# B&R Automation Studio project NAEUL004C00R13L518F00 (part 35)

#### Act_Main.st - Do Not Change!!!
```iecst
(** 2022-12-20 **)
ACTION Act_Background:

	a_tyAlmData[1]	:= tyAlmData;

	IF (bRstErr = TRUE) THEN

		tylocalAlm.Out.bErr		:= FALSE;
		tylocalAlm.Out.bWarning	:= FALSE;

		//Reset Warning
		memset(ADR(a_tyWarningCurrList) , 0 , SIZEOF(a_tyWarningCurrList));
		udiWarningMax	:=1;

		memset(ADR(tylocalAlm.Out.a_tyCurrList) , 0 , SIZEOF(tylocalAlm.Out.a_tyCurrList));
	//	memset(ADR(tylocalAlm.Out.a_sRecoveryList) , 0 , SIZEOF(tylocalAlm.Out.a_sRecoveryList));
		memset(ADR(tylocalAlm.Out.a_udiRecoveryList),0,SIZEOF(tylocalAlm.Out.a_udiRecoveryList));

		udiAlmCntr	:= 0;

		bAlmUpdt	:= FALSE;

	END_IF

	IF (bRstWarning = TRUE) THEN

		IF tylocalAlm.Out.bErr =FALSE AND tylocalAlm.Out.bWarning= TRUE THEN
			//Reset Warning
			memset(ADR(a_tyWarningCurrList) , 0 , SIZEOF(a_tyWarningCurrList));
			udiWarningMax	:=1;

			memset(ADR(tylocalAlm.Out.a_tyCurrList) , 0 , SIZEOF(tylocalAlm.Out.a_tyCurrList));
		//	memset(ADR(tylocalAlm.Out.a_sRecoveryList) , 0 , SIZEOF(tylocalAlm.Out.a_sRecoveryList));
			memset(ADR(tylocalAlm.Out.a_udiRecoveryList),0,SIZEOF(tylocalAlm.Out.a_udiRecoveryList));
			udiAlmCntr	:= 0;
			tylocalAlm.Out.bWarning := FALSE;
		END_IF

		bAlmUpdt	:= FALSE;

	END_IF

	IF bAlarmLog = TRUE  AND tylocalAlm.In.bStartupUISettingsLoadDone THEN

		IF (bAlmUpdt = FALSE) OR (tylocalAlm.Out.eStatus = Error) THEN

			tylocalAlm.Out.bInfo		:= FALSE;
			tylocalAlm.Out.bInfoLF		:= FALSE;
			iInfoCntr	:= 0;

			FOR udi := 1 TO c_udiAlarmCurrMax DO

				IF (a_tyAlmData[udi].udiRunTime <> a_udiRunTimeOld[udi]) AND a_tyAlmData[udi].udiCode <> 0
					AND ((a_tyAlmData[udi].eSeverity = AlmSeverityError ) ) THEN

					a_udiRunTimeOld[udi]	:= a_tyAlmData[udi].udiRunTime;

					bAlmUpdt	:= TRUE;

					udiAlmCntr	:= udiAlmCntr + 1;
					IF udiAlmCntr > c_udiAlarmCurrMax THEN
						udiAlmCntr	:= c_udiAlarmCurrMax;
					END_IF

					udiLogCntr	:= udiLogCntr + 1;
					IF udiLogCntr > c_udiAlarmCurrMax THEN
						udiLogCntr	:= c_udiAlarmCurrMax;
					END_IF

					fLogDTConvert(ADR(sDT) , tylocalAlm.In.dtCurrDT);

					IF a_tyAlmData[udi].udiCode < 10000 THEN
						udiErrorCode := a_tyAlmData[udi].udiCode;
					ELSE
						udiErrorCode := (a_tyAlmData[udi].udiCode - 10000) + (a_tyAlmData[udi].udiModuleNum);//*For HMI Text Group*
					END_IF

					//In this case, Program Name/Data Time/
					//Current List
					tylocalAlm.Out.a_tyCurrList[udiAlmCntr].eSeverity		:= a_tyAlmData[udi].eSeverity;
					tylocalAlm.Out.a_tyCurrList[udiAlmCntr].sDT				:= sDT;

					//To HMI Text Group
					tylocalAlm.Out.a_tyCurrList[udiAlmCntr].udiErrorCode	:= udiErrorCode;
					tylocalAlm.Out.a_tyCurrList[udiAlmCntr].bAlm			:= a_tyAlmData[udi].bAlm;

					//Recovery List
					tylocalAlm.Out.a_udiRecoveryList[udiAlmCntr]			:= udiErrorCode; //*For HMI Text Group **It will be the same procedure with the above**

					//History List
					memmove(ADR(a_tyHistoryList[2]) , ADR(a_tyHistoryList[1]) , SIZEOF(a_tyHistoryList[1]) * (c_udiAlarmHistoryMax - 1));

					a_tyHistoryList[1].sDT				:= sDT;
					a_tyHistoryList[1].udiModErrCode	:= a_tyAlmData[udi].udiCode;
					a_tyHistoryList[1].udiErrorCode		:= udiErrorCode;

					//Log List
					//					fLogAlmDispMsg(ADR(sAlmMsg) , tylocalAlm.In.dtCurrDT , a_tyAlmData[udi].sProgNm , a_tyAlmData[udi].udiCode , a_tyAlmData[udi].sAlmMsg); // *For Log files*
					//					a_sLogList[udiLogCntr]	:= sAlmMsg;
					a_sLogList[udiLogCntr]	:= CONCAT(a_sLogList[udiLogCntr] , '$r$n');

					//Severity
					IF a_tyAlmData[udi].eSeverity = AlmSeverityError THEN
						tylocalAlm.Out.bErr		:= TRUE;
					END_IF

					// Alarm warning
				ELSIF (( a_tyAlmData[udi].eSeverity = AlmSeverityWarning) AND  (a_tyAlmData[udi].udiCode <> 0 )) THEN

					//Used to compare
					memset(ADR(sWarningCompareMsg) , 0 , SIZEOF(sWarningCompareMsg));

					//					sWarningCompareMsg	:= CONCAT(sWarningCompareMsg , a_tyAlmData[udi].sProgNm);
					//					sWarningCompareMsg	:= CONCAT(sWarningCompareMsg , ' | ');
					//					sWarningID := UDINT_TO_STRING(a_tyAlmData[udi].udiCode);
					//					sWarningCompareMsg	:= CONCAT(sWarningCompareMsg , sWarningID);
					//					sWarningCompareMsg	:= CONCAT(sWarningCompareMsg , ' | ');
					////					sWarningCompareMsg	:= CONCAT(sWarningCompareMsg , a_tyAlmData[udi].sAlmMsg);
					//
					//					//Checking whether it is recorded in the alarm list
					//					FOR udi1 := 0 TO  udiWarningMax DO
					//						WarningListOccur := (memcmp(ADR(sWarningCompareMsg),ADR(a_tyWarningCurrList[udi1].sMsg),SIZEOF(sWarningCompareMsg) )= 0);
					//
					//						IF WarningListOccur THEN
					//							EXIT;
					//						END_IF
					//
					//					END_FOR

					//IF warning message is no recorded in alarm list
					IF 	WarningListOccur =FALSE THEN

						bAlmUpdt	:= TRUE;
						udiWarningMax := udiWarningMax +1;

						udiAlmCntr	:= udiAlmCntr + 1;

						IF udiAlmCntr > c_udiAlarmCurrMax THEN
							udiAlmCntr	:= c_udiAlarmCurrMax;
						END_IF

						udiRecorded[udiWarningMax-1]:= udi;

						udiLogCntr	:= udiLogCntr + 1;

						IF udiLogCntr > c_udiAlarmCurrMax THEN
							udiLogCntr	:= c_udiAlarmCurrMax;
						END_IF

						//Warning List
						//						a_tyWarningCurrList[udiWarningMax-1].sMsg		:= sWarningCompareMsg;

						fLogDTConvert(ADR(sDT) , tylocalAlm.In.dtCurrDT);
						udiErrorCode := (a_tyAlmData[udi].udiCode - 10000) + a_tyAlmData[udi].udiModuleNum; //*For HMI Text Group*

						//Current List
						tylocalAlm.Out.a_tyCurrList[udiAlmCntr].eSeverity		:= a_tyAlmData[udi].eSeverity;
						tylocalAlm.Out.a_tyCurrList[udiAlmCntr].sDT				:= sDT;
						tylocalAlm.Out.a_tyCurrList[udiAlmCntr].udiModErrCode	:= a_tyAlmData[udi].udiCode;

						//To HMI Text Group
						tylocalAlm.Out.a_tyCurrList[udiAlmCntr].udiErrorCode	:= udiErrorCode;
						tylocalAlm.Out.a_tyCurrList[udiAlmCntr].bWarning		:= a_tyAlmData[udi].bWarning;

						//Recovery List
						//						tylocalAlm.Out.a_sRecoveryList[udiAlmCntr]	 	:= a_tyAlmData[udi].sRcyMsg;
						tylocalAlm.Out.a_udiRecoveryList[udiAlmCntr]	:= udiErrorCode;

						//History List
						memmove(ADR(a_tyHistoryList[2]) , ADR(a_tyHistoryList[1]) , SIZEOF(a_tyHistoryList[1]) * (c_udiAlarmHistoryMax - 1));

						a_tyHistoryList[1].sDT				:= sDT;
						a_tyHistoryList[1].udiModErrCode	:= a_tyAlmData[udi].udiCode;
						a_tyHistoryList[1].udiErrorCode		:= udiErrorCode;

						//Log List
						//Info Message
						//						fLogAlmDispMsg(ADR(sWarningMsg) , tylocalAlm.In.dtCurrDT , a_tyAlmData[udi].sProgNm , a_tyAlmData[udi].udiCode , a_tyAlmData[udi].sAlmMsg);

						a_sLogList[udiLogCntr]	:= sWarningMsg;
						a_sLogList[udiLogCntr]	:= CONCAT(a_sLogList[udiLogCntr] , '$r$n');

						tylocalAlm.Out.bWarning	:= TRUE;

					END_IF

					// Show Info Message
				ELSIF  ((a_tyAlmData[udi].udiCode <> 0) AND (a_tyAlmData[udi].eSeverity = AlmSeverityInfo)) THEN

					iInfoCntr	:= iInfoCntr + 1;

					IF iInfoCntr = 1 THEN

						IF a_tyAlmData[udi].udiModuleNum = 3901 AND a_tyAlmData[udi].bAlm THEN //Identify Leader Follower Inforamtion

							tylocalAlm.Out.bInfoLF	:= TRUE;
							tylocalAlm.Out.bInfo	:= TRUE;

						ELSE
							tylocalAlm.Out.bInfoLF	:= FALSE;
							tylocalAlm.Out.bInfo	:= TRUE;
						END_IF

					ELSIF iInfoCntr = 2 THEN
						//						tylocalAlm.sInfoMsg	:= CONCAT(tylocalAlm.sInfoMsg , '$r$n$r$n');
						//						tylocalAlm.sInfoMsg	:= CONCAT(tylocalAlm.sInfoMsg , a_tyAlmData[udi].sAlmMsg);

					END_IF

				END_IF

			END_FOR

		ELSE

			tylocalAlm.In.eAct	:= AlarmActAppendLogWriteHistory;
			IF tylocalAlm.Out.eStatus = Done AND tylocalAlm.Out.eStat = AlarmActAppendLogWriteHistory THEN
				tylocalAlm.In.eAct		:= AlarmActIdle;
				bAlmUpdt	:= FALSE;
				udiLogCntr	:= 0;
			END_IF

		END_IF

	END_IF
	//**** Background Running Done*****

	//Delete Old Alarm Log File for 24 hours After Machine is Continuous Running 30 Days.
	fbDlyTmr(IN := TRUE);
	IF fbDlyTmr.Q THEN
		fbDeleteLogTmr (IN := TRUE);
		IF fbDeleteLogTmr.Q AND eStatus <> Busy THEN
			p_eAct := AlarmActDeleteOldLog;
			IF eStat = AlarmActDeleteOldLog AND eStatus = Done THEN
				p_eAct := AlarmActIdle;
				fbDlyTmr (IN := FALSE);
				fbDeleteLogTmr (IN := FALSE);
			END_IF
		END_IF
	END_IF

	//Reset Done
	IF tylocalAlm.Out.eStatus = Done AND tylocalAlm.In.eAct = AlarmActIdle THEN
		tylocalAlm.Out.eStat	:= AlarmActIdle;
	END_IF

	//Set tylocalAlm.In.eAct
	IF tylocalAlm.Out.eStatus = Idle THEN
		tylocalAlm.Out.eStat	:= tylocalAlm.In.eAct;
	END_IF
	//Main
	CASE tylocalAlm.Out.eStat OF

		AlarmActIdle:
			IF tylocalAlm.Out.eStatus <> Idle THEN	//Reset Data
				//Private
				fbDirCreate1(bEn := FALSE);
				fbDirCreate2(bEn := FALSE);
				fbFileOldDel1(bEn := FALSE);
				fbFileRead1(bEn := FALSE);
				fbFileAppend1(bEn := FALSE);
				fbFileWrite1(bEn := FALSE);
				usiStep	:= 0;

				tylocalAlm.Out.bHistoryFileNotFound	:= FALSE;
				udiWriteLogCntr			:= 1;

				sStatTxt	:= a_sStatText[tylocalAlm.Out.eStat];

			END_IF

			tylocalAlm.Out.eStatus	:= Idle;

		AlarmActCreateDir:
			IF tylocalAlm.Out.eStatus = Idle OR tylocalAlm.Out.eStatus = Busy THEN

				tylocalAlm.Out.eStatus	:= Busy;

				sStatTxt	:= a_sStatText[tylocalAlm.Out.eStat];

				CASE usiStep OF
					0:
						fbDirCreate1(bEn := TRUE);
						IF fbDirCreate1.udiStatus = 0 THEN
							usiStep	:= 1;
						ELSIF fbDirCreate1.udiStatus < 65534 THEN
							tylocalAlm.Out.eStatus		:= Error;

							IF fbDirCreate1.udiStatus = 1908 THEN
								udiStatus	:= 5051;	//Create User Directory Error
							ELSE
								udiStatus	:= fbDirCreate1.udiStatus;
							END_IF
						END_IF

					1:
						fbDirCreate2(bEn := TRUE);
						IF fbDirCreate2.udiStatus = 0 THEN
							tylocalAlm.Out.eStatus	:= Done;
						ELSIF fbDirCreate2.udiStatus < 65534 THEN
							tylocalAlm.Out.eStatus		:= Error;

							IF fbDirCreate2.udiStatus = 1908 THEN
								udiStatus	:= 5052;	//Create Alarm Directory Error
							ELSE
								udiStatus	:= fbDirCreate2.udiStatus;
							END_IF
						END_IF

				END_CASE

			END_IF

		AlarmActDeleteOldLog:
			IF tylocalAlm.Out.eStatus = Idle OR tylocalAlm.Out.eStatus = Busy THEN

				tylocalAlm.Out.eStatus	:= Busy;

				sStatTxt	:= a_sStatText[tylocalAlm.Out.eStat];

				fbFileOldDel1.dtDTNow			:= tylocalAlm.In.dtCurrDT;
				fbFileOldDel1.udiFileKeepDay	:= tylocalAlm.In.udiFileKeepDay;
				fbFileOldDel1(bEn := TRUE);
				IF fbFileOldDel1.udiStatus = 0 THEN
					tylocalAlm.Out.eStatus	:= Done;
				ELSIF fbFileOldDel1.udiStatus < 65534 THEN
					tylocalAlm.Out.eStatus		:= Error;

					IF fbFileOldDel1.udiStatus = 1910 THEN
						udiStatus	:= 5053;	//Get Directory Info Error While Deleting Old Log
					ELSIF fbFileOldDel1.udiStatus = 1911 THEN
						udiStatus	:= 5054;	//Directory Read Error While Deleting Old Log
					ELSIF fbFileOldDel1.udiStatus = 1912 THEN
						udiStatus	:= 5055;	//File Delete Error While Deleting Old Log
					ELSE
						udiStatus	:= fbFileOldDel1.udiStatus;
					END_IF
				END_IF

			END_IF

		AlarmActReadHistory:
			IF tylocalAlm.Out.eStatus = Idle OR tylocalAlm.Out.eStatus = Busy THEN

				tylocalAlm.Out.eStatus	:= Busy;

				sStatTxt	:= a_sStatText[tylocalAlm.Out.eStat];

				fbFileRead1(bEn := TRUE);
				IF fbFileRead1.udiStatus = 0 THEN
					tylocalAlm.Out.eStatus	:= Done;
				ELSIF fbFileRead1.udiStatus < 65534 THEN
					tylocalAlm.Out.eStatus		:= Error;

					IF fbFileRead1.udiStatus = 1900 THEN
						udiStatus	:= 5056;	//File Open Error While Reading Alarm History
					ELSIF fbFileRead1.udiStatus = 1902 THEN
						udiStatus	:= 5057;	//File Read Error While Reading Alarm History
					ELSIF fbFileRead1.udiStatus = 1904 THEN
						udiStatus	:= 5058;	//File Close Error While Reading Alarm History
					ELSIF fbFileRead1.udiStatus = 1915 THEN
						tylocalAlm.Out.eStatus					:= Done;
						tylocalAlm.Out.bHistoryFileNotFound	:= TRUE;
					ELSE
						udiStatus	:= fbFileRead1.udiStatus;
					END_IF
				END_IF

			END_IF

		AlarmActWriteHistory:
			IF tylocalAlm.Out.eStatus = Idle OR tylocalAlm.Out.eStatus = Busy THEN

				tylocalAlm.Out.eStatus	:= Busy;

				sStatTxt	:= a_sStatText[tylocalAlm.Out.eStat];

				fbFileWrite1(bEn := TRUE);
				IF fbFileWrite1.udiStatus = 0 THEN
					tylocalAlm.Out.eStatus	:= Done;
				ELSIF fbFileWrite1.udiStatus < 65534 THEN
					tylocalAlm.Out.eStatus		:= Error;

					IF fbFileWrite1.udiStatus = 1900 THEN
						udiStatus	:= 5059;	//File Open Error While Writing Alarm History
					ELSIF fbFileWrite1.udiStatus = 1901 THEN
						udiStatus	:= 5060;	//File Create Error While Writing Alarm History
					ELSIF fbFileWrite1.udiStatus = 1903 THEN
						udiStatus	:= 5061;	//File Write Error While Writing Alarm History
					ELSIF fbFileWrite1.udiStatus = 1904 THEN
						udiStatus	:= 5062;	//File Close Error While Writing Alarm History
					ELSIF fbFileWrite1.udiStatus = 1914 THEN
						udiStatus	:= 5063;	//Directory Does Not Exist While Writing Alarm History
					ELSE
						udiStatus	:= fbFileWrite1.udiStatus;
					END_IF
				END_IF

			END_IF

		AlarmActAppendLog:
			IF tylocalAlm.Out.eStatus = Idle OR tylocalAlm.Out.eStatus = Busy THEN

				tylocalAlm.Out.eStatus	:= Busy;

				sStatTxt	:= a_sStatText[tylocalAlm.Out.eStat];

				dtCurrDTTemp			:= tylocalAlm.In.dtCurrDT;
				fbFileAppend1.sFile		:= DT_TO_STRING(dtCurrDTTemp);
				fbFileAppend1.sFile		:= MID(fbFileAppend1.sFile , 10 , 4);
				fbFileAppend1.sFile		:= CONCAT('ALARM_' , fbFileAppend1.sFile);
				fbFileAppend1.sFile		:= CONCAT(fbFileAppend1.sFile , '.dat');

				fbFileAppend1.p_Src		:= ADR(a_sLogList[udiWriteLogCntr]);
				fbFileAppend1.udiLen	:= LEN(a_sLogList[udiWriteLogCntr]);

				fbFileAppend1(bEn := TRUE);
				IF fbFileAppend1.udiStatus = 0 THEN
					IF udiWriteLogCntr >= udiLogCntr THEN
						tylocalAlm.Out.eStatus	:= Done;
					ELSE
						udiWriteLogCntr	:= udiWriteLogCntr + 1;
						fbFileAppend1(bEn := FALSE);
					END_IF

				ELSIF fbFileAppend1.udiStatus < 65534 THEN
					tylocalAlm.Out.eStatus		:= Error;

					IF fbFileAppend1.udiStatus = 1900 THEN
						udiStatus	:= 5064;	//File Open Error While Writing Alarm Log
					ELSIF fbFileAppend1.udiStatus = 1901 THEN
						udiStatus	:= 5065;	//File Create Error While Writing Alarm Log
					ELSIF fbFileAppend1.udiStatus = 1913 THEN
						udiStatus	:= 5066;	//Get File Info Error While Writing Alarm Log
					ELSIF fbFileAppend1.udiStatus = 1903 THEN
						udiStatus	:= 5067;	//File Write Error While Writing Alarm Log
					ELSIF fbFileAppend1.udiStatus = 1904 THEN
						udiStatus	:= 5068;	//File Close Error While Writing Alarm Log
					ELSIF fbFileAppend1.udiStatus = 1914 THEN
						udiStatus	:= 5069;	//Directory Does Not Exist While Writing Alarm Log
					ELSE
						udiStatus	:= fbFileAppend1.udiStatus;
					END_IF
				END_IF

			END_IF

		AlarmActAppendLogWriteHistory:
			IF tylocalAlm.Out.eStatus = Idle OR tylocalAlm.Out.eStatus = Busy THEN

				tylocalAlm.Out.eStatus	:= Busy;

				sStatTxt	:= a_sStatText[tylocalAlm.Out.eStat];

				dtCurrDTTemp			:= tylocalAlm.In.dtCurrDT;
				fbFileAppend1.sFile		:= DT_TO_STRING(dtCurrDTTemp);
				fbFileAppend1.sFile		:= MID(fbFileAppend1.sFile , 10 , 4);
				fbFileAppend1.sFile		:= CONCAT('ALARM_' , fbFileAppend1.sFile);
				fbFileAppend1.sFile		:= CONCAT(fbFileAppend1.sFile , '.dat');

				fbFileAppend1.p_Src		:= ADR(a_sLogList[udiWriteLogCntr]);
				fbFileAppend1.udiLen	:= LEN(a_sLogList[udiWriteLogCntr]);

				fbFileAppend1(bEn := TRUE);
				fbFileWrite1(bEn := TRUE);

				IF (fbFileAppend1.udiStatus = 0) AND (udiWriteLogCntr >= udiLogCntr) AND fbFileWrite1.udiStatus = 0 THEN
					tylocalAlm.Out.eStatus	:= Done;

				ELSIF fbFileAppend1.udiStatus = 0 AND udiWriteLogCntr < udiLogCntr THEN
					udiWriteLogCntr	:= udiWriteLogCntr + 1;
					fbFileAppend1(bEn := FALSE);

				ELSIF fbFileWrite1.udiStatus > 0 AND fbFileWrite1.udiStatus < 65534 THEN
					tylocalAlm.Out.eStatus		:= Error;

					IF fbFileWrite1.udiStatus = 1900 THEN
						udiStatus	:= 5070;	//File Open Error While Writing Alarm History
					ELSIF fbFileWrite1.udiStatus = 1901 THEN
						udiStatus	:= 5071;	//File Create Error While Writing Alarm History
					ELSIF fbFileWrite1.udiStatus = 1903 THEN
						udiStatus	:= 5072;	//File Write Error While Writing Alarm History
					ELSIF fbFileWrite1.udiStatus = 1904 THEN
						udiStatus	:= 5073;	//File Close Error While Writing Alarm History
					ELSIF fbFileWrite1.udiStatus = 1914 THEN
						udiStatus	:= 5074;	//Directory Does Not Exist While Writing Alarm History
					ELSE
						udiStatus	:= fbFileWrite1.udiStatus;
					END_IF

				ELSIF fbFileAppend1.udiStatus > 0 AND fbFileAppend1.udiStatus < 65534 THEN
					tylocalAlm.Out.eStatus		:= Error;

					IF fbFileAppend1.udiStatus = 1900 THEN
						udiStatus	:= 5075;	//File Open Error While Writing Alarm Log
					ELSIF fbFileAppend1.udiStatus = 1901 THEN
						udiStatus	:= 5076;	//File Create Error While Writing Alarm Log
					ELSIF fbFileAppend1.udiStatus = 1913 THEN
						udiStatus	:= 5077;	//Get File Info Error While Writing Alarm Log
					ELSIF fbFileAppend1.udiStatus = 1903 THEN
						udiStatus	:= 5078;	//File Write Error While Writing Alarm Log
					ELSIF fbFileAppend1.udiStatus = 1904 THEN
						udiStatus	:= 5079;	//File Close Error While Writing Alarm Log
					ELSIF fbFileAppend1.udiStatus = 1914 THEN
						udiStatus	:= 5080;	//Directory Does Not Exist While Writing Alarm Log
					ELSE
						udiStatus	:= fbFileAppend1.udiStatus;
					END_IF
				END_IF

			END_IF

		AlarmActResetHistory:
			IF tylocalAlm.Out.eStatus = Idle OR tylocalAlm.Out.eStatus = Busy THEN

				tylocalAlm.Out.eStatus	:= Busy;

				sStatTxt	:= a_sStatText[tylocalAlm.Out.eStat];

				memset(ADR(a_tyHistoryList) , 0 , SIZEOF(a_tyHistoryList));

				fbFileWrite1(bEn := TRUE);
				IF fbFileWrite1.udiStatus = 0 THEN
					tylocalAlm.Out.eStatus	:= Done;
				ELSIF fbFileWrite1.udiStatus < 65534 THEN
					tylocalAlm.Out.eStatus		:= Error;

					IF fbFileWrite1.udiStatus = 1900 THEN
						udiStatus	:= 5081;	//File Open Error While Resetting Alarm History
					ELSIF fbFileWrite1.udiStatus = 1901 THEN
						udiStatus	:= 5082;	//File Create Error While Resetting Alarm History
					ELSIF fbFileWrite1.udiStatus = 1903 THEN
						udiStatus	:= 5083;	//File Write Error While Resetting Alarm History
					ELSIF fbFileWrite1.udiStatus = 1904 THEN
						udiStatus	:= 5084;	//File Close Error While Resetting Alarm History
					ELSIF fbFileWrite1.udiStatus = 1914 THEN
						udiStatus	:= 5085;	//Directory Does Not Exist While Resetting Alarm History
					ELSE
						udiStatus	:= fbFileWrite1.udiStatus;
					END_IF
				END_IF

			END_IF

		AlarmActBGStartLog:
			IF tylocalAlm.Out.eStatus = Idle OR tylocalAlm.Out.eStatus = Busy THEN

				sStatTxt	:= a_sStatText[tylocalAlm.Out.eStat];

				bAlarmLog	:= TRUE;
				tylocalAlm.Out.eStatus		:= Done;

			END_IF

		AlarmActBGStopLog:
			IF tylocalAlm.Out.eStatus = Idle OR tylocalAlm.Out.eStatus = Busy THEN

				sStatTxt	:= a_sStatText[tylocalAlm.Out.eStat];

				bAlarmLog	:= FALSE;
				tylocalAlm.Out.eStatus		:= Done;

			END_IF

	END_CASE

	END_CASE
END_ACTION
```

#### Act_Alarm.st - Do Not Change!!!
```iecst
(** 2019-03-25 **)
ACTION Act_Alarm:
	IF tylocalAlm.In.udiRstErr <> udiRstErrOld THEN
		bRstErr			:= TRUE;
		udiRstErrOld	:= tylocalAlm.In.udiRstErr;
	ELSE
		bRstErr			:= FALSE;
	END_IF

	//Checking which Warning is clear
	IF a_tyWarningCurrList[1].sMsg <> '' AND p_tyLinkLibVerAlmData.udiCode = 0 THEN

		FOR udi2 := 1 TO (udiWarningMax-1) DO
			udiRecorded1:= udiRecorded[udi2];
			IF 	(pa_tyAlmData[udiRecorded1].eSeverity =  AlmSeverityNA) AND udiRecorded1<> 0 THEN
				bRstWarning := TRUE;
				EXIT;
			ELSE
				bRstWarning := FALSE;
			END_IF

		END_FOR
	ELSE
		bRstWarning := FALSE;
	END_IF

	//Reset Error
	IF (tylocalAlm.Out.eStatus = Error) AND bRstErr THEN
		tylocalAlm.In.eAct	:= AlarmActIdle;
		tylocalAlm.Out.eStat	:= AlarmActIdle;
	END_IF

	//Error
	IF EDGEPOS(tylocalAlm.Out.eStatus = Error) THEN

		tyAlmData.udiCode				:= udiStatus;
		tyAlmData.eSeverity				:= AlmSeverityError;
		tyAlmData.udiRunTime			:= tyAlmData.udiRunTime + 1;
		tyAlmData.bAlm					:= TRUE;
		tyAlmData.udiModuleNum  		:= udiModuleNum;
		g_tyAlmProgNm.sAlarmProgNm		:= g_tyNtParamCurr.sAlmProgNm;

		//Get Error Message
		IF tyAlmData.udiCode < 10000 OR tyAlmData.udiCode > 10099 THEN
			tyAlmData.sAlmMsg	:= 'Unknown';
			tyAlmData.sRcyMsg	:= 'Unknown';
		ELSE
			tyAlmData.sAlmMsg	:= a_tyAlmText[tyAlmData.udiCode].sAlmText;
			tyAlmData.sRcyMsg	:= a_tyAlmText[tyAlmData.udiCode].sRcyText;
		END_IF

		sStatTxt	:= tyAlmData.sAlmMsg;
	ELSIF bRstErr AND (tyAlmData.udiCode <> 0) THEN

		tyAlmData.udiCode	:= 0;
		tyAlmData.eSeverity	:= AlmSeverityNA;
		tyAlmData.bAlm			:= FALSE;
		sStatTxt	:= a_sStatText[tylocalAlm.Out.eStat];

	END_IF

END_ACTION
```

#### InputRef.var - Do Not Change!!!
```iecst
(*2019-03-25*)
(**)
(*General*)
VAR
	p_udiCurrMax : REFERENCE TO UDINT;
	p_udiHistoryMax : REFERENCE TO UDINT;
END_VAR
(**)
VAR
	p_eAct : REFERENCE TO eAlarmAction;
	p_udiRstErr : REFERENCE TO UDINT;
END_VAR
(**)
(*Configuration*)
VAR
	p_dtCurrDT : REFERENCE TO DATE_AND_TIME;
	pa_tyAlmData : REFERENCE TO ARRAY[1..c_udiAlarmCurrMax] OF tyAlmDat;
	p_udiFileKeepDay : REFERENCE TO UDINT;
	p_sProgNm : REFERENCE TO STRING[15];
	p_bNtSettingsLoadDone : REFERENCE TO BOOL;
	p_bStartupUISettingsLoadDone : REFERENCE TO BOOL;
END_VAR
```

#### Local.var - Do Not Change!!!
```iecst
(*2019-05-09*)
(**)
(*Local Action, State & Status*)
VAR
	udiStatus : UDINT := 0;
	sStatTxt : STRING[200] := '';
	a_sStatText : ARRAY[0..50] OF STRING[200] := ['Idling','Creating Directory','Deleting Old Alarm Log File','Reading History File','Writing History File','Appending Alarm Log File','Appending Alarm Log File & Writing History File','Resetting History','Background Start Alarm Log','Background Stop Alarm Log',41('')];
END_VAR
(**)
(*Local Alarm*)
VAR
	tyAlmData : tyAlmDat;
	tylocalAlm : tyAlarm;
	a_tyAlmData : ARRAY[1..c_udiAlarmCurrMax] OF tyAlmDat;
END_VAR
(**)
(*Local Output*)
VAR
	bErr : BOOL;
	bWarning : BOOL;
	a_tyCurrList : ARRAY[1..c_udiAlarmCurrMax] OF tyAlarmCurr;
	a_udiRecoveryList : ARRAY[1..c_udiAlarmCurrMax] OF UDINT;
	a_sHistoryList : ARRAY[1..c_udiAlarmHistoryMax] OF STRING[200];
	bInfo : BOOL;
	sInfoMsg : STRING[200];
	bHistoryFileNotFound : BOOL;
	bInfoLF : BOOL := FALSE;
END_VAR
(**)
(*Local Input*)
VAR
	udiRstErr : UDINT := 0;
	dtCurrDT : DATE_AND_TIME;
	udiFileKeepDay : UDINT := 30;
	sProgNm : STRING[15] := 'Alarm';
	bNtSettingsLoadDone : BOOL := TRUE;
END_VAR
(**)
(*Local*)
VAR
	bRstErr : BOOL;
	udiRstErrOld : UDINT;
	bInitDone : BOOL;
	bInitialDone : BOOL;
	bAlarmLog : BOOL;
	usiStep : USINT;
	udi : UDINT;
	iInfoCntr : INT;
	sAlmMsg : STRING[300];
	udiAlmCntr : UDINT;
	udiAlmRecvryCntr : UDINT;
	udiLogCntr : UDINT;
	udiWriteLogCntr : UDINT;
	a_sLogList : ARRAY[1..c_udiAlarmCurrMax] OF STRING[200];
	bAlmUpdt : BOOL;
	dtCurrDTTemp : DATE_AND_TIME;
	a_udiRunTimeOld : ARRAY[1..c_udiAlarmCurrMax] OF UDINT;
	fbDirCreate1 : fbDirCreate;
	fbDirCreate2 : fbDirCreate;
	fbFileAppend1 : fbFileFullAppend;
	fbFileOldDel1 : fbFileOldDel;
	fbFileRead1 : fbFileFullRead;
	fbFileWrite1 : fbFileFullWrite;
	udi1 : UDINT;
	udi2 : UDINT;
	udiRecorded : ARRAY[1..c_udiAlarmCurrMax] OF UDINT;
	udiRecorded1 : UDINT;
	bRstWarning : BOOL;
	udiWarningMax : UDINT := 1;
	sWarningMsg : STRING[300];
	sWarningID : STRING[80] := '';
	sWarningCompareMsg : STRING[300];
	a_tyWarningCurrList : ARRAY[1..c_udiAlarmCurrMax] OF tyAlarmCurr;
	a_tyHistoryList : ARRAY[1..c_udiAlarmHistoryMax] OF tyHistory;
	WarningListOccur : BOOL := TRUE;
	udiErrorCode : UDINT;
	sDT : STRING[80];
	sLogString : STRING[200];
	udiModuleNum : UDINT := 5051;
END_VAR
```

#### Act_InputConfig.st - not listed in the package file held
```iecst
ACTION Act_InputConfig:

	tylocalAlm.In.udiRstErr					 := g_tyRstErrOut.udiRstErr;
	tylocalAlm.In.eAct					 	 := g_tyStartUp.eAlarmAct;
	tylocalAlm.In.dtCurrDT  			  	 := g_tyTime.dtCurrDT;
	tylocalAlm.In.udiFileKeepDay		 	 := g_tyNtParamCurr.udiAlmFileKeepDay;
	tylocalAlm.In.sProgNm					 := g_tyNtParamCurr.sAlmProgNm;
	tylocalAlm.In.bStartupUISettingsLoadDone := g_tyStartUp.bUISettingsLoadDone;

	//Index 1 For Internal Use
	a_tyAlmData[2]		:= g_tyUsrFolder.tyAlmData;
	a_tyAlmData[3]		:= g_tyLibVer.tyAlmData;
	a_tyAlmData[4]		:= g_tyTime.tyAlmData;
	a_tyAlmData[5]		:= g_tyTime.tyAlmData1;
	a_tyAlmData[6]		:= g_tyHWInfo.tyAlmData;
	a_tyAlmData[7]		:= g_tyProdRcp.tyAlmData;
	a_tyAlmData[8]		:= g_tyMpProdRcp.tyAlmData;
	a_tyAlmData[9]		:= g_tyMagRcp.tyAlmData;
	a_tyAlmData[10]		:= g_tyMcParam.tyAlmData;
	a_tyAlmData[11]		:= g_tyNtParam.tyAlmData;
	a_tyAlmData[12]		:= g_tyUsrMgmt.tyAlmData;
	a_tyAlmData[13]		:= g_tyBuffer1.tyAlmData;
	a_tyAlmData[14]		:= g_tyBuffer2.tyAlmData;
	a_tyAlmData[15]		:= g_tyBuffer3.tyAlmData;
	a_tyAlmData[16]		:= g_tyUSSMEMAA.tyAlmData;
	a_tyAlmData[17]		:= g_tyUSSMEMAB.tyAlmData;
	a_tyAlmData[18]		:= g_tyUSSMEMA1.tyAlmData;
	a_tyAlmData[19]		:= g_tyUSSMEMA2.tyAlmData;
	a_tyAlmData[20]		:= g_tyUSSMEMA3.tyAlmData;
	a_tyAlmData[21]		:= g_tyDSSMEMA1.tyAlmData;
	a_tyAlmData[22]		:= g_tyDSSMEMA2.tyAlmData;
	a_tyAlmData[23]		:= g_tyDSSMEMA3.tyAlmData;
	a_tyAlmData[24]		:= g_tyInShutter.tyAlmData;
	a_tyAlmData[25]		:= g_tyOutShutter.tyAlmData;
	a_tyAlmData[26]		:= g_tyStopperA.tyAlmData;
	a_tyAlmData[27]		:= g_tyStopperB.tyAlmData;
	a_tyAlmData[28]		:= g_tyPshrConv.tyAlmData;
	a_tyAlmData[29]		:= g_tyMagConv1.tyAlmData;
	a_tyAlmData[30]		:= g_tyMagConv2.tyAlmData;
	a_tyAlmData[31]		:= g_tyMagConv3.tyAlmData;
	a_tyAlmData[32]	:= g_tyAWOpen.tyAlmData;
	a_tyAlmData[33]	:= g_tyAWOpen.tyAlmData1;
	a_tyAlmData[34]	:= g_tyAWOpen.tyAlmData2;
	a_tyAlmData[35]	:= g_tyAWOpen.tyAlmData3;
	a_tyAlmData[36]	:= g_tyTrav.tyAlmData;
	a_tyAlmData[37]	:= g_tyTrav.tyAlmData1;
	a_tyAlmData[38]	:= g_tyTrav.tyAlmData2;
	a_tyAlmData[39]	:= g_tyTrav.tyAlmData3;
	a_tyAlmData[40]	:= g_tyLifterBtm.tyAlmData;
	a_tyAlmData[41]	:= g_tyLifterBtm.tyAlmData1;
	a_tyAlmData[42]	:= g_tyLifterBtm.tyAlmData2;
	a_tyAlmData[43]	:= g_tyLifterBtm.tyAlmData3;
	a_tyAlmData[44]	:= g_tyDI.tyAlmData1;
	a_tyAlmData[45]	:= g_tyDI.tyAlmData2;
	a_tyAlmData[46]	:= g_tyDI.tyAlmData3;
	a_tyAlmData[47]	:= g_tyDI.tyAlmData4;
	a_tyAlmData[48]	:= g_tyAGVMag1.tyAlmData;
	a_tyAlmData[49]	:= g_tyAGVMag2.tyAlmData;
	a_tyAlmData[50]	:= g_tyAGVMag3.tyAlmData;
	a_tyAlmData[51]	:= g_tyHermes.tyAlmData;
	a_tyAlmData[52]	:= g_tyUSHermesA.tyAlmData;
	a_tyAlmData[53]	:= g_tyUSHermesA.tyAlmData1;
	a_tyAlmData[54]	:= g_tyUSHermesA.tyAlmData2;
	a_tyAlmData[55]	:= g_tyUSHermesA.tyAlmData3;
	a_tyAlmData[56]	:= g_tyUSHermesA.tyAlmData4;
	a_tyAlmData[57]	:= g_tyUSHermesAInfoData;
	a_tyAlmData[58]	:= g_tyUSHermesB.tyAlmData;
	a_tyAlmData[59]	:= g_tyUSHermesB.tyAlmData1;
	a_tyAlmData[60]	:= g_tyUSHermesB.tyAlmData2;
	a_tyAlmData[61]	:= g_tyUSHermesB.tyAlmData3;
	a_tyAlmData[62]	:= g_tyUSHermesB.tyAlmData4;
	a_tyAlmData[63]	:= g_tyUSHermesBInfoData;
	a_tyAlmData[64]	:= g_tyRmtHermes.tyAlmData;
	a_tyAlmData[65]	:= g_tyRmtHermes.tyAlmData1;
	a_tyAlmData[66]	:= g_tyRmtHermes.tyAlmData2;
	a_tyAlmData[67]	:= g_tyRmtHermes.tyAlmData3;
	a_tyAlmData[68]	:= g_tyLFLeader.tyAlmData;
	a_tyAlmData[69]	:= g_tyLFFollower.tyAlmData;
	a_tyAlmData[70]	:= g_tyLFFollowerInfoData;
	a_tyAlmData[71]	:= g_tyLFFollowerInfoData1;
	a_tyAlmData[72]	:= g_tyFollower1.tyAlmData;
	a_tyAlmData[73]	:= g_tyFollower1InfoData;
	a_tyAlmData[74]	:= g_tyFollower1InfoData1;
	a_tyAlmData[75]	:= g_tyFollower2.tyAlmData;
	a_tyAlmData[76]	:= g_tyFollower2InfoData;
	a_tyAlmData[77]	:= g_tyFollower2InfoData1;
	a_tyAlmData[78]	:= g_tyLCSMngRcp.tyAlmData;
	a_tyAlmData[79]	:= g_tyLCSLF.tyAlmData;
	a_tyAlmData[80]	:= g_tyLCSLFInfoData;
	a_tyAlmData[81]	:= g_tyOpsTravLifUL.tyAlmData;
	//	a_tyAlmData[82]	:= g_tyOpsMagUL1.tyAlmData;
	//	a_tyAlmData[83]	:= g_tyOpsMagUL1.tyAlmData1;
	//	a_tyAlmData[84]	:= g_tyOpsMagUL2.tyAlmData;
	//	a_tyAlmData[85]	:= g_tyOpsMagUL2.tyAlmData1;
	//	a_tyAlmData[86]	:= g_tyOpsMagUL3.tyAlmData;
	//	a_tyAlmData[87]	:= g_tyOpsMagUL3.tyAlmData1;
	a_tyAlmData[82]	:= g_tyOpsLifMagUL.tyAlmData;
	a_tyAlmData[83]	:= g_tyOpsLifMagUL.tyAlmData1;
	a_tyAlmData[84]	:= g_tyOpsLifMagUL.tyAlmData2;

	a_tyAlmData[88]	:= g_tyOpsMagConvUL1.tyAlmData;
	a_tyAlmData[89]	:= g_tyOpsMagConvUL1.tyAlmData1;
	a_tyAlmData[90]	:= g_tyOpsMagConvUL2.tyAlmData;
	a_tyAlmData[91]	:= g_tyOpsMagConvUL2.tyAlmData1;
	a_tyAlmData[92]	:= g_tyOpsMagConvUL3.tyAlmData;
	a_tyAlmData[93]	:= g_tyOpsMagConvUL3.tyAlmData1;
	a_tyAlmData[94]	:= g_tyUSHermesA.tyAlmData5;
	a_tyAlmData[95]	:= g_tyUSHermesB.tyAlmData5;
	a_tyAlmData[96]	:= g_tyMcAlarmData;
	a_tyAlmData[97]	:= g_tyMag1SafetyBar.tyAlmData;
	a_tyAlmData[98]	:= g_tyMag2SafetyBar.tyAlmData;
	a_tyAlmData[99]	:= g_tyMag3SafetyBar.tyAlmData;
	a_tyAlmData[100]	:= g_tyMag1AWEngage.tyAlmData;
	a_tyAlmData[101]	:= g_tyMag2AWEngage.tyAlmData;
	a_tyAlmData[102]	:= g_tyMag3AWEngage.tyAlmData;
	a_tyAlmData[103]	:= g_tyMag1SafetyBar.tyAlmData;
	a_tyAlmData[104]	:= g_tyMag2SafetyBar.tyAlmData;
	a_tyAlmData[105]	:= g_tyMag3SafetyBar.tyAlmData;
	a_tyAlmData[106]	:= g_tyMag1AWEngage.tyAlmData;
	a_tyAlmData[107]	:= g_tyMag2AWEngage.tyAlmData;
	a_tyAlmData[108]	:= g_tyMag3AWEngage.tyAlmData;
	a_tyAlmData[109]	:= g_tyMagAWOpen1.tyAlmData;
	a_tyAlmData[110]	:= g_tyMagAWOpen1.tyAlmData1;
	a_tyAlmData[111]	:= g_tyMagAWOpen1.tyAlmData2;
	a_tyAlmData[112]	:= g_tyMagAWOpen1.tyAlmData3;
	a_tyAlmData[113]	:= g_tyMagAWOpen2.tyAlmData;
	a_tyAlmData[114]	:= g_tyMagAWOpen2.tyAlmData1;
	a_tyAlmData[115]	:= g_tyMagAWOpen2.tyAlmData2;
	a_tyAlmData[116]	:= g_tyMagAWOpen2.tyAlmData3;
	a_tyAlmData[117]	:= g_tyMagAWOpen3.tyAlmData;
	a_tyAlmData[118]	:= g_tyMagAWOpen3.tyAlmData1;
	a_tyAlmData[119]	:= g_tyMagAWOpen3.tyAlmData2;
	a_tyAlmData[120]	:= g_tyMagAWOpen3.tyAlmData3;
	a_tyAlmData[121]	:= g_tyMcAlarmData;
	a_tyAlmData[122]	:= g_tyUSSOT1.tyAlmData;
	a_tyAlmData[123]	:= g_tyUSSOT2.tyAlmData;
	a_tyAlmData[124]	:= g_tyUSSOT3.tyAlmData;
	a_tyAlmData[125]	:= g_tyDSSOT1.tyAlmData;
	a_tyAlmData[126]	:= g_tyDSSOT2.tyAlmData;
	a_tyAlmData[127]	:= g_tyDSSOT3.tyAlmData;
	a_tyAlmData[128]	:= g_tyMag1SelClamp.tyAlmData;
	a_tyAlmData[129]	:= g_tyMag2SelClamp.tyAlmData;
	a_tyAlmData[130]	:= g_tyMag3SelClamp.tyAlmData;
	a_tyAlmData[131]	:= g_tyAWPushOrPuller.tyAlmData;
	a_tyAlmData[132]	:= g_tyAWPushOrPuller.tyAlmData1;
	a_tyAlmData[133]	:= g_tyAWPushOrPuller.tyAlmData2;
	a_tyAlmData[134]	:= g_tyAWPushOrPuller.tyAlmData3;
	a_tyAlmData[135]	:= g_tyMtrPshr.tyAlmData;
	a_tyAlmData[136]	:= g_tyAGV.tyAlmData1;
	a_tyAlmData[150]	:= g_tyDI.tyAlmData5;

	IF g_tyNtParamCurr.bProjMagConvLane1Prep AND g_tyNtParamCurr.bProjMagConvLane2Prep THEN
		a_tyAlmData[167]	:= g_tyOpsInMagConv.tyAlmData;
		a_tyAlmData[168]	:= g_tyOpsOutMagConv.tyAlmData;
	END_IF
	IF g_tyNtParamCurr.bProjMagConvLane1Prep THEN //customized
		a_tyAlmData[151]	:= g_tyTopEntStpr.tyAlmData; //MagConv Lane1
		a_tyAlmData[152]	:= g_tyTopMidStpr.tyAlmData;
		a_tyAlmData[153]	:= g_tyTopExtStpr.tyAlmData;
		a_tyAlmData[154]	:= g_tyBtmMidStpr.tyAlmData;
		a_tyAlmData[155]	:= g_tyBtmExtStpr.tyAlmData;
		a_tyAlmData[161]	:= g_tyInMagConv.tyAlmData;
		a_tyAlmData[162]	:= g_tyOutMagConv.tyAlmData;
		a_tyAlmData[165]	:= g_tyLifterMagConv.tyAlmData;
	END_IF
	IF  g_tyNtParamCurr.bProjMagConvLane2Prep  THEN
		a_tyAlmData[156]	:= g_tyTopEntStpr2.tyAlmData; //MagConv Lane2
		a_tyAlmData[157]	:= g_tyTopMidStpr2.tyAlmData;
		a_tyAlmData[158]	:= g_tyTopExtStpr2.tyAlmData;
		a_tyAlmData[159]	:= g_tyBtmMidStpr2.tyAlmData;
		a_tyAlmData[160]	:= g_tyBtmExtStpr2.tyAlmData;
		a_tyAlmData[163]	:= g_tyInMagConv2.tyAlmData;
		a_tyAlmData[164]	:= g_tyOutMagConv2.tyAlmData;
		a_tyAlmData[166]	:= g_tyLifterMagConv2.tyAlmData;
	END_IF
	IF g_tyNtParamCurr.bProjLifter2Prep THEN
		a_tyAlmData[169]	:= g_tyLifter2.tyAlmData;
		a_tyAlmData[170]	:= g_tyLifter2.tyAlmData1;
		a_tyAlmData[171]	:= g_tyLifter2.tyAlmData2;
		a_tyAlmData[172]	:= g_tyLifter2.tyAlmData3;
	END_IF
	a_tyAlmData[173]	:= g_tyPP.tyAlmData;
	a_tyAlmData[174]	:= g_tyPP.tyAlmData1;
	a_tyAlmData[175]	:= g_tyPP.tyAlmData2;
	a_tyAlmData[176]	:= g_tyPP.tyAlmData3;
	a_tyAlmData[177]	:= g_tyDI.tyAlmData6;
	a_tyAlmData[178]	:= g_tyOutShutter.tyAlmData2;
	a_tyAlmData[179]	:= g_tyOutShutter.tyAlmData3;
	IF g_tyNtParamCurr.bProjTCPAGVSigPrep THEN
		a_tyAlmData[180]	:= g_tyTCP.tyAlmData;
		a_tyAlmData[181]	:= g_tyTCP.tyAlmData1;
		a_tyAlmData[182]	:= g_tyTCP.tyAlmData2;
		a_tyAlmData[183]	:= g_tyTCP.tyAlmData3;
	END_IF
	IF g_tyNtParamCurr.bProjScanPrep THEN
		a_tyAlmData[184]	:= g_tyTCPTop.tyAlmData;
		a_tyAlmData[185]	:= g_tyTCPBtm.tyAlmData;
	END_IF

	a_tyAlmData[186] := g_tySvyHermes.tyAlmData;
	a_tyAlmData[187] := g_tySvyHermes.tyAlmData1;
	a_tyAlmData[188] := g_tySvyHermes.tyAlmData2;
	a_tyAlmData[189] := g_tySvyHermes.tyAlmData3;
	a_tyAlmData[190] := g_tySvyHermes.tyAlmData4;
	a_tyAlmData[191] := g_tySvyHermesInfoData;
	a_tyAlmData[192] := g_tySvyHermesInfoData1;
	a_tyAlmData[193] := g_tySvyHermesInfoData2;
	a_tyAlmData[194] := g_tySvyHermesInfoData3;
	a_tyAlmData[195] := g_tySvyHermesInfoDat;

	IF g_tyNtParamCurr.bAutoRcpPrep THEN
		a_tyAlmData[195] :=  g_tyAutoRcp.tyAlmData;
	END_IF

END_ACTION
```

#### Act_OutputConfig.st - not listed in the package file held
```iecst
ACTION Act_OutputConfig:

	g_tyAlm := tylocalAlm.Out;

END_ACTION
```

### RstErr.typ - Do Not Change!!!
```iecst
TYPE
	eRstErrAction :
		(
		RstErrActIdle,
		RstErrActRun,
		RstErrActSetSafetyRlyRst,
		RstErrActRstSafetyRlyRst
		);
	tyRstErrIn1 : 	STRUCT
		eAct : eRstErrAction; (*Reset Error's Action*)
		bSafetyRlySig : BOOL; (*Safety Relay Signal*)
		bManual : BOOL := FALSE; (*Manual Mode*)
	END_STRUCT;
	tyRstErrOut1 : 	STRUCT
		eStat : eRstErrAction := RstErrActIdle; (*Reset Error's State*)
		eStatus : eFBStatus := Idle; (*Reset Error's Status*)
		sStatTxt : STRING[200] := ''; (*Reset Error's State in Text*)
		udiRstErr : UDINT; (*Reset Error*)
		bSafetyRlyRst : BOOL; (*Safety Relay Reset*)
	END_STRUCT;
	tyRstErr : 	STRUCT
		In : tyRstErrIn1;
		Out : tyRstErrOut1;
	END_STRUCT;
END_TYPE
```

### RstErr.var - Change By Project
```iecst
VAR
	g_tyRstErrOut : tyRstErrOut1;
END_VAR
```

### Program Logical/RstErr/RstErr (IEC, version 1.00.0) - 1.00.0 - 

#### Act_InputConfig.st - Change By Project
```iecst
ACTION Act_InputConfig:

// Input Configuration - Others
 tylocalRstErr.In.eAct          := g_tyUIOut.eMnlAct.eRstErrAct;
 tylocalRstErr.In.bSafetyRlySig := g_tyDInput.bSafetyRlySig;

END_ACTION
```

#### Act_OutputConfig.st - Change By Project
```iecst
ACTION Act_OutputConfig:

	g_tyRstErrOut := tylocalRstErr.Out;

END_ACTION
```

#### Cyclic.st - Do Not Change!!!
```iecst
PROGRAM _CYCLIC

	IF bInitialDone = FALSE THEN
		IF g_tyStartUp.bNtSettingsLoadDone = TRUE THEN
			bInitialDone	:= TRUE;
			Act_Initial;
		END_IF

	ELSE
		Act_InputConfig;
		Act_Main;
		Act_OutputConfig;

	END_IF

END_PROGRAM
```

#### Act_Initial.st - Do Not Change!!!
```iecst
ACTION Act_Initial:

	//Initial
	tylocalRstErr.Out.sStatTxt	:= a_sStatText[tylocalRstErr.Out.eStat];

	fbSafetyRlyRstTm(IN := FALSE);

END_ACTION
```

#### Act_Main.st - Do Not Change!!!
```iecst
ACTION Act_Main:

	IF EDGENEG(tylocalRstErr.In.bManual) THEN
		tylocalRstErr.In.eAct	:= RstErrActIdle;
	END_IF

	//Reset Done
	IF tylocalRstErr.Out.eStatus = Done AND tylocalRstErr.In.eAct = RstErrActIdle THEN
		tylocalRstErr.Out.eStat	:= RstErrActIdle;
	END_IF

	//Set p_eAct
	IF tylocalRstErr.Out.eStatus = Idle THEN
		tylocalRstErr.Out.eStat	:= tylocalRstErr.In.eAct;
	END_IF

	//Main
	CASE tylocalRstErr.Out.eStat OF

		RstErrActIdle:
			IF tylocalRstErr.Out.eStatus <> Idle THEN	//Reset Data
				//Private
				fbSafetyRlyRstTm(IN := FALSE);

				tylocalRstErr.Out.sStatTxt	:= a_sStatText[tylocalRstErr.Out.eStat];

				IF tylocalRstErr.In.bManual = FALSE THEN
					tylocalRstErr.Out.bSafetyRlyRst	:= FALSE;
				END_IF

			END_IF

			IF EDGENEG(tylocalRstErr.In.bManual) THEN
				tylocalRstErr.Out.bSafetyRlyRst	:= FALSE;
			END_IF

			tylocalRstErr.Out.eStatus	:= Idle;

		RstErrActRun:
			IF tylocalRstErr.Out.eStatus = Idle OR tylocalRstErr.Out.eStatus = Busy THEN

				tylocalRstErr.Out.eStatus	:= Busy;

				tylocalRstErr.Out.sStatTxt	:= a_sStatText[tylocalRstErr.Out.eStat];

				IF tylocalRstErr.Out.bSafetyRlyRst=FALSE THEN
					tylocalRstErr.Out.udiRstErr	:= tylocalRstErr.Out.udiRstErr + 1;
				END_IF

				IF tylocalRstErr.In.bSafetyRlySig = FALSE THEN
					tylocalRstErr.Out.bSafetyRlyRst	:= TRUE;
				END_IF

				IF tylocalRstErr.Out.bSafetyRlyRst = TRUE THEN
					fbSafetyRlyRstTm(IN := TRUE, PT := T#500ms);

					IF fbSafetyRlyRstTm.Q = TRUE THEN
						tylocalRstErr.Out.bSafetyRlyRst	:= FALSE;
						tylocalRstErr.Out.eStatus			:= Done;
					END_IF

				ELSE
					tylocalRstErr.Out.eStatus	:= Done;

				END_IF

			END_IF

		RstErrActSetSafetyRlyRst:
			IF tylocalRstErr.Out.eStatus = Idle OR tylocalRstErr.Out.eStatus = Busy THEN

				tylocalRstErr.Out.sStatTxt	:= a_sStatText[tylocalRstErr.Out.eStat];

				//Reset
				fbSafetyRlyRstTm(IN := FALSE);

				tylocalRstErr.Out.bSafetyRlyRst	:= TRUE;
				tylocalRstErr.Out.eStatus			:= Done;

			END_IF

		RstErrActRstSafetyRlyRst:
			IF tylocalRstErr.Out.eStatus = Idle OR tylocalRstErr.Out.eStatus = Busy THEN

				tylocalRstErr.Out.sStatTxt	:= a_sStatText[tylocalRstErr.Out.eStat];

				//Reset
				fbSafetyRlyRstTm(IN := FALSE);

				tylocalRstErr.Out.bSafetyRlyRst	:= FALSE;
				tylocalRstErr.Out.eStatus			:= Done;

			END_IF

	END_CASE

END_ACTION
```

#### Local.var - Do Not Change!!!
```iecst
VAR
	eAct : eRstErrAction := RstErrActIdle;
	eStatus : eFBStatus := Idle;
	sStatTxt : STRING[200] := '';
	a_sStatText : ARRAY[0..50] OF STRING[200] := ['Idling','Running Reset Error','Turning On Safety Relay Reset','Turning Off Safety Relay Reset',47('')];
END_VAR
(**)
(*Local Alarm*)
(**)
(*Local Output*)
VAR
	udiRstErr : UDINT;
	bSafetyRlyRst : BOOL;
END_VAR
(**)
(*Local Input*)
VAR
	bManual : BOOL := FALSE;
	bSafetyRlySig : BOOL;
	bNtSettingsLoadDone : BOOL := TRUE;
END_VAR
(**)
(*Local*)
VAR
	bInitDone : BOOL;
	bInitialDone : BOOL;
	fbSafetyRlyRstTm : TON;
	tylocalRstErr : tyRstErr;
END_VAR
```

### ProdRcp.typ - Change By Project
```iecst
(*2020-07-24*)
(**)
(*Action*)

TYPE
	eProdRcpAction :
		(
		ProdRcpActIdle,
		ProdRcpActCreateDir,
		ProdRcpActAddEdit,
		ProdRcpActDel,
		ProdRcpActGetInfo,
		ProdRcpActGetList,
		ProdRcpActFilter,
		ProdRcpActLoadRcp,
		ProdRcpActAdd,
		ProdRcpActEdit,
		ProdRcpActReadCurrRcp,
		ProdRcpActWriteCurrRcpParam,
		ProdRcpActSaveList,
		ProdRcpActSort,
		ProdRcpActEndCharFilter
		);
END_TYPE

(**)
(*Data*)

TYPE
	tyProdRcpParam : 	STRUCT
		sRcpNm : STRING[254];
		diWidthInUM : DINT;
		diWidthInUM2 : DINT;
		diIntvlCntr : DINT;
		diMinSltValue : DINT;
		diMaxSltValue : DINT;
		diPitch : DINT;
		diBrdPerSlt : DINT;
		usiMcMod : USINT;
		bTopToBtm : BOOL;
		bGapBwtnBrd : BOOL;
		bLongBrd : BOOL;
		diMinReqFreeBffr : DINT;
		sDisplayInfo : STRING[30];
		dtLastModified : DATE_AND_TIME;
		diMtrPshrExtSpd : DINT;
		diMtrPshrExtTorq : DINT;
		diPshrOffset : DINT;
	END_STRUCT;
	tyProdRcpIn1 : 	STRUCT
		udiRstErr : UDINT;
		sSearch : STRING[254];
		sScan : STRING[254];
		tyInfoIn : tyProdRcpParam;
		tyCurrRcpWr : tyProdRcpParam;
		sProgNm : STRING[15];
		bWidth2Prep : BOOL;
	END_STRUCT;
	tyProdRcpOut1 : 	STRUCT
		eStat : eProdRcpAction;
		eStatus : eFBStatus;
		sStatTxt : STRING[200];
		tyAlmData : tyAlmDat;
	END_STRUCT;
	tyProdRcp : 	STRUCT
		In : tyProdRcpIn1;
		Out : tyProdRcpOut1;
	END_STRUCT;
END_TYPE
```

### ProdRcp.var - Change By Project
```iecst
(**)
(*Constant*)
VAR CONSTANT
	c_udiProdRcpMax : UDINT := 2000;
END_VAR
VAR
	g_tyProdRcp : tyProdRcpOut1;
END_VAR
(**)
(*Alarm*)
VAR
	p_ProdRcpAlmData : UDINT;
END_VAR
(**)
(*Output*)
VAR
	p_ProdRcpNmExist : UDINT;
	p_ProdRcpNmNotExist : UDINT;
	p_ProdRcpNmEmpty : UDINT;
	p_ProdRcpListFull : UDINT;
	p_ProdRcpCurrList : UDINT;
	p_ProdRcpFilterList : UDINT;
	p_ProdRcpSortedList : UDINT;
	p_ProdRcpScanList : UDINT;
	p_ProdRcpInfoOut : UDINT;
	p_ProdRcpFileNotFound : UDINT;
	p_ProdRcpCurrRcpAll : UDINT;
END_VAR
(**)
VAR
	p_ProdRcpCurrRcp0 : UDINT;
	p_ProdRcpCurrRcp0Nm : UDINT;
	p_ProdRcpCurrRcp0Width : UDINT;
	p_ProdRcpCurrRcp0MinSltValue : UDINT;
	p_ProdRcpCurrRcp0MaxSltValue : UDINT;
	p_ProdRcpCurrRcp0Pitch : UDINT;
	p_ProdRcpCurrRcp0BrdPerSlt : UDINT;
	p_ProdRcpCurrRcp0McMod : UDINT;
	p_ProdRcpCurrRcp0TopToBtm : UDINT;
	p_ProdRcpCurrRcp0GapBtwnBrd : UDINT;
	p_ProdRcpCurrRcp0LongBrd : UDINT;
	p_ProdRcpCurrRcp0MinReqFreeBffr : UDINT;
	p_ProdRcpCurrRcp0DisplayInfo : UDINT;
	p_ProdRcpCurrRcp0LastModified : UDINT;
	p_ProdRcpCurrRcp0Width2 : UDINT;
	p_ProdRcpCurrRcp0PshrPulerOffset : UDINT;
	p_ProdRcpCurrRcp0MtrPshrExtSpd : UDINT;
	p_ProdRcpCurrRcp0MtrPshrExtTorq : UDINT;
	p_ProdRcpCurrRcp0PshrOffset : UDINT;
END_VAR
(**)
VAR
	p_ProdRcpCurrRcp1 : UDINT;
	p_ProdRcpCurrRcp1Nm : UDINT;
	p_ProdRcpCurrRcp1Width : UDINT;
	p_ProdRcpCurrRcp1MinSltValue : UDINT;
	p_ProdRcpCurrRcp1MaxSltValue : UDINT;
	p_ProdRcpCurrRcp1Pitch : UDINT;
	p_ProdRcpCurrRcp1BrdPerSlt : UDINT;
	p_ProdRcpCurrRcp1McMod : UDINT;
	p_ProdRcpCurrRcp1TopToBtm : UDINT;
	p_ProdRcpCurrRcp1GapBtwnBrd : UDINT;
	p_ProdRcpCurrRcp1LongBrd : UDINT;
	p_ProdRcpCurrRcp1MinReqFreeBffr : UDINT;
	p_ProdRcpCurrRcp1DisplayInfo : UDINT;
	p_ProdRcpCurrRcp1LastModified : UDINT;
	p_ProdRcpCurrRcp1Width2 : UDINT;
	p_ProdRcpCurrRcp1PshrPulerOffset : UDINT;
	p_ProdRcpCurrRcp1MtrPshrExtSpd : UDINT;
	p_ProdRcpCurrRcp1MtrPshrExtTorq : UDINT;
	p_ProdRcpCurrRcp1PshrOffset : UDINT;
END_VAR
(**)
VAR
	p_ProdRcpCurrRcp2 : UDINT;
	p_ProdRcpCurrRcp2Nm : UDINT;
	p_ProdRcpCurrRcp2Width : UDINT;
	p_ProdRcpCurrRcp2MinSltValue : UDINT;
	p_ProdRcpCurrRcp2MaxSltValue : UDINT;
	p_ProdRcpCurrRcp2Pitch : UDINT;
	p_ProdRcpCurrRcp2BrdPerSlt : UDINT;
	p_ProdRcpCurrRcp2McMod : UDINT;
	p_ProdRcpCurrRcp2TopToBtm : UDINT;
	p_ProdRcpCurrRcp2GapBtwnBrd : UDINT;
	p_ProdRcpCurrRcp2LongBrd : UDINT;
	p_ProdRcpCurrRcp2MinReqFreeBffr : UDINT;
	p_ProdRcpCurrRcp2DisplayInfo : UDINT;
	p_ProdRcpCurrRcp2LastModified : UDINT;
	p_ProdRcpCurrRcp2Width2 : UDINT;
	p_ProdRcpCurrRcp2PshrPulerOffset : UDINT;
	p_ProdRcpCurrRcp2MtrPshrExtSpd : UDINT;
	p_ProdRcpCurrRcp2MtrPshrExtTorq : UDINT;
	p_ProdRcpCurrRcp2PshrOffset : UDINT;
END_VAR
(**)
VAR
	p_ProdRcpCurrRcp3 : UDINT;
	p_ProdRcpCurrRcp3Nm : UDINT;
	p_ProdRcpCurrRcp3Width : UDINT;
	p_ProdRcpCurrRcp3MinSltValue : UDINT;
	p_ProdRcpCurrRcp3MaxSltValue : UDINT;
	p_ProdRcpCurrRcp3Pitch : UDINT;
	p_ProdRcpCurrRcp3BrdPerSlt : UDINT;
	p_ProdRcpCurrRcp3McMod : UDINT;
	p_ProdRcpCurrRcp3TopToBtm : UDINT;
	p_ProdRcpCurrRcp3GapBtwnBrd : UDINT;
	p_ProdRcpCurrRcp3LongBrd : UDINT;
	p_ProdRcpCurrRcp3MinReqFreeBffr : UDINT;
	p_ProdRcpCurrRcp3DisplayInfo : UDINT;
	p_ProdRcpCurrRcp3LastModified : UDINT;
	p_ProdRcpCurrRcp3Width2 : UDINT;
	p_ProdRcpCurrRcp3PshrPulerOffset : UDINT;
	p_ProdRcpCurrRcp3MtrPshrExtSpd : UDINT;
	p_ProdRcpCurrRcp3MtrPshrExtTorq : UDINT;
	p_ProdRcpCurrRcp3PshrOffset : UDINT;
END_VAR
(**)
VAR
	p_ProdRcpCurrRcp4 : UDINT;
	p_ProdRcpCurrRcp4Nm : UDINT;
	p_ProdRcpCurrRcp4Width : UDINT;
	p_ProdRcpCurrRcp4MinSltValue : UDINT;
	p_ProdRcpCurrRcp4MaxSltValue : UDINT;
	p_ProdRcpCurrRcp4Pitch : UDINT;
	p_ProdRcpCurrRcp4BrdPerSlt : UDINT;
	p_ProdRcpCurrRcp4McMod : UDINT;
	p_ProdRcpCurrRcp4TopToBtm : UDINT;
	p_ProdRcpCurrRcp4GapBtwnBrd : UDINT;
	p_ProdRcpCurrRcp4LongBrd : UDINT;
	p_ProdRcpCurrRcp4MinReqFreeBffr : UDINT;
	p_ProdRcpCurrRcp4DisplayInfo : UDINT;
	p_ProdRcpCurrRcp4LastModified : UDINT;
	p_ProdRcpCurrRcp4Width2 : UDINT;
	p_ProdRcpCurrRcp4PshrPulerOffset : UDINT;
	p_ProdRcpCurrRcp4MtrPshrExtSpd : UDINT;
	p_ProdRcpCurrRcp4MtrPshrExtTorq : UDINT;
	p_ProdRcpCurrRcp4PshrOffset : UDINT;
END_VAR
(**)
VAR
	p_ProdRcpCurrRcp5 : UDINT;
	p_ProdRcpCurrRcp5Nm : UDINT;
	p_ProdRcpCurrRcp5Width : UDINT;
	p_ProdRcpCurrRcp5MinSltValue : UDINT;
	p_ProdRcpCurrRcp5MaxSltValue : UDINT;
	p_ProdRcpCurrRcp5Pitch : UDINT;
	p_ProdRcpCurrRcp5BrdPerSlt : UDINT;
	p_ProdRcpCurrRcp5McMod : UDINT;
	p_ProdRcpCurrRcp5TopToBtm : UDINT;
	p_ProdRcpCurrRcp5GapBtwnBrd : UDINT;
	p_ProdRcpCurrRcp5LongBrd : UDINT;
	p_ProdRcpCurrRcp5MinReqFreeBffr : UDINT;
	p_ProdRcpCurrRcp5DisplayInfo : UDINT;
	p_ProdRcpCurrRcp5LastModified : UDINT;
	p_ProdRcpCurrRcp5Width2 : UDINT;
	p_ProdRcpCurrRcp5PshrPulerOffset : UDINT;
	p_ProdRcpCurrRcp5MtrPshrExtSpd : UDINT;
	p_ProdRcpCurrRcp5MtrPshrExtTorq : UDINT;
	p_ProdRcpCurrRcp5PshrOffset : UDINT;
END_VAR
(**)
```

### Program Logical/ProdRcp/ProdRcp (IEC, version 1.00.0) - 1.00.0 - NtRecipe v5.00.0 , NtFileIO v5.00.0

#### Init.st - Change By Project
```iecst
(** 2020-06-08 **)
PROGRAM _INIT

	(* Always Change If Project Change *)

	//Pass Address To Global Address For External Use
	//Action, State & Status
	p_ProdRcpStat		:= ADR(eStat);
	p_ProdRcpStatus		:= ADR(eStatus);
	p_ProdRcpStatTxt	:= ADR(sStatTxt);

	//Alarm
	p_ProdRcpAlmData	:= ADR(tyAlmData);

	//Output
	p_ProdRcpNmExist		:= ADR(bNmExist);
	p_ProdRcpNmNotExist		:= ADR(bNmNotExist);
	p_ProdRcpNmEmpty		:= ADR(bNmEmpty);
	p_ProdRcpListFull		:= ADR(bListFull);
	p_ProdRcpCurrList		:= ADR(a_tyCurrList);
	p_ProdRcpFilterList		:= ADR(a_tyFilterList);
	p_ProdRcpSortedList				:= ADR(a_tySortList);
	p_ProdRcpScanList				:= ADR(a_tyScanList);
	p_ProdRcpInfoOut		:= ADR(tyInfoOut);
	p_ProdRcpFileNotFound	:= ADR(bFileNotFound);
	p_ProdRcpCurrRcpAll		:= ADR(a_tyCurrRcp);
	p_ProdRcpCurrRcp0				:= ADR(a_tyCurrRcp[0]);
	p_ProdRcpCurrRcp0Nm				:= ADR(a_tyCurrRcp[0].sRcpNm);
	p_ProdRcpCurrRcp0Width			:= ADR(a_tyCurrRcp[0].diWidthInUM);
	p_ProdRcpCurrRcp0MinSltValue	:= ADR(a_tyCurrRcp[0].diMinSltValue);
	p_ProdRcpCurrRcp0MaxSltValue	:= ADR(a_tyCurrRcp[0].diMaxSltValue);
	p_ProdRcpCurrRcp0Pitch			:= ADR(a_tyCurrRcp[0].diPitch);
	p_ProdRcpCurrRcp0BrdPerSlt		:= ADR(a_tyCurrRcp[0].diBrdPerSlt);
	p_ProdRcpCurrRcp0McMod			:= ADR(a_tyCurrRcp[0].usiMcMod);
	p_ProdRcpCurrRcp0TopToBtm		:= ADR(a_tyCurrRcp[0].bTopToBtm);
	p_ProdRcpCurrRcp0GapBtwnBrd		:= ADR(a_tyCurrRcp[0].bGapBwtnBrd);
	p_ProdRcpCurrRcp0LongBrd		:= ADR(a_tyCurrRcp[0].bLongBrd);
	p_ProdRcpCurrRcp0MinReqFreeBffr	:= ADR(a_tyCurrRcp[0].diMinReqFreeBffr);
	p_ProdRcpCurrRcp0DisplayInfo	:= ADR(a_tyCurrRcp[0].sDisplayInfo);
	p_ProdRcpCurrRcp0LastModified	:= ADR(a_tyCurrRcp[0].dtLastModified);
	p_ProdRcpCurrRcp0Width2 		:= ADR(a_tyCurrRcp[0].diWidthInUM2);
	p_ProdRcpCurrRcp0PshrPulerOffset:= ADR(a_tyCurrRcp[0].diPshrOffset);
	p_ProdRcpCurrRcp0MtrPshrExtSpd	:= ADR(a_tyCurrRcp[0].diMtrPshrExtSpd);
	p_ProdRcpCurrRcp0MtrPshrExtTorq	:= ADR(a_tyCurrRcp[0].diMtrPshrExtTorq);
	p_ProdRcpCurrRcp0PshrOffset		:= ADR(a_tyCurrRcp[0].diPshrOffset);

	p_ProdRcpCurrRcp1				:= ADR(a_tyCurrRcp[1]);
	p_ProdRcpCurrRcp1Nm				:= ADR(a_tyCurrRcp[1].sRcpNm);
	p_ProdRcpCurrRcp1Width			:= ADR(a_tyCurrRcp[1].diWidthInUM);
	p_ProdRcpCurrRcp1MinSltValue	:= ADR(a_tyCurrRcp[1].diMinSltValue);
	p_ProdRcpCurrRcp1MaxSltValue	:= ADR(a_tyCurrRcp[1].diMaxSltValue);
	p_ProdRcpCurrRcp1Pitch			:= ADR(a_tyCurrRcp[1].diPitch);
	p_ProdRcpCurrRcp1BrdPerSlt		:= ADR(a_tyCurrRcp[1].diBrdPerSlt);
	p_ProdRcpCurrRcp1McMod			:= ADR(a_tyCurrRcp[1].usiMcMod);
	p_ProdRcpCurrRcp1TopToBtm		:= ADR(a_tyCurrRcp[1].bTopToBtm);
	p_ProdRcpCurrRcp1GapBtwnBrd		:= ADR(a_tyCurrRcp[1].bGapBwtnBrd);
	p_ProdRcpCurrRcp1LongBrd		:= ADR(a_tyCurrRcp[1].bLongBrd);
	p_ProdRcpCurrRcp1MinReqFreeBffr	:= ADR(a_tyCurrRcp[1].diMinReqFreeBffr);
	p_ProdRcpCurrRcp1DisplayInfo	:= ADR(a_tyCurrRcp[1].sDisplayInfo);
	p_ProdRcpCurrRcp1LastModified	:= ADR(a_tyCurrRcp[1].dtLastModified);
	p_ProdRcpCurrRcp1Width2 		:= ADR(a_tyCurrRcp[1].diWidthInUM2);
	p_ProdRcpCurrRcp1PshrPulerOffset:= ADR(a_tyCurrRcp[1].diPshrOffset);
	p_ProdRcpCurrRcp1MtrPshrExtSpd	:= ADR(a_tyCurrRcp[1].diMtrPshrExtSpd);
	p_ProdRcpCurrRcp1MtrPshrExtTorq	:= ADR(a_tyCurrRcp[1].diMtrPshrExtTorq);
	p_ProdRcpCurrRcp1PshrOffset		:= ADR(a_tyCurrRcp[1].diPshrOffset);

	p_ProdRcpCurrRcp2				:= ADR(a_tyCurrRcp[2]);
	p_ProdRcpCurrRcp2Nm				:= ADR(a_tyCurrRcp[2].sRcpNm);
	p_ProdRcpCurrRcp2Width			:= ADR(a_tyCurrRcp[2].diWidthInUM);
	p_ProdRcpCurrRcp2MinSltValue	:= ADR(a_tyCurrRcp[2].diMinSltValue);
	p_ProdRcpCurrRcp2MaxSltValue	:= ADR(a_tyCurrRcp[2].diMaxSltValue);
	p_ProdRcpCurrRcp2Pitch			:= ADR(a_tyCurrRcp[2].diPitch);
	p_ProdRcpCurrRcp2BrdPerSlt		:= ADR(a_tyCurrRcp[2].diBrdPerSlt);
	p_ProdRcpCurrRcp2McMod			:= ADR(a_tyCurrRcp[2].usiMcMod);
	p_ProdRcpCurrRcp2TopToBtm		:= ADR(a_tyCurrRcp[2].bTopToBtm);
	p_ProdRcpCurrRcp2GapBtwnBrd		:= ADR(a_tyCurrRcp[2].bGapBwtnBrd);
	p_ProdRcpCurrRcp2LongBrd		:= ADR(a_tyCurrRcp[2].bLongBrd);
	p_ProdRcpCurrRcp2MinReqFreeBffr	:= ADR(a_tyCurrRcp[2].diMinReqFreeBffr);
	p_ProdRcpCurrRcp2DisplayInfo	:= ADR(a_tyCurrRcp[2].sDisplayInfo);
	p_ProdRcpCurrRcp2LastModified	:= ADR(a_tyCurrRcp[2].dtLastModified);
	p_ProdRcpCurrRcp2Width2 		:= ADR(a_tyCurrRcp[2].diWidthInUM2);
	p_ProdRcpCurrRcp2PshrPulerOffset:= ADR(a_tyCurrRcp[2].diPshrOffset);
	p_ProdRcpCurrRcp2MtrPshrExtSpd	:= ADR(a_tyCurrRcp[2].diMtrPshrExtSpd);
	p_ProdRcpCurrRcp2MtrPshrExtTorq	:= ADR(a_tyCurrRcp[2].diMtrPshrExtTorq);
	p_ProdRcpCurrRcp2PshrOffset		:= ADR(a_tyCurrRcp[2].diPshrOffset);

	p_ProdRcpCurrRcp3				:= ADR(a_tyCurrRcp[3]);
	p_ProdRcpCurrRcp3Nm				:= ADR(a_tyCurrRcp[3].sRcpNm);
	p_ProdRcpCurrRcp3Width			:= ADR(a_tyCurrRcp[3].diWidthInUM);
	p_ProdRcpCurrRcp3MinSltValue	:= ADR(a_tyCurrRcp[3].diMinSltValue);
	p_ProdRcpCurrRcp3MaxSltValue	:= ADR(a_tyCurrRcp[3].diMaxSltValue);
	p_ProdRcpCurrRcp3Pitch			:= ADR(a_tyCurrRcp[3].diPitch);
	p_ProdRcpCurrRcp3BrdPerSlt		:= ADR(a_tyCurrRcp[3].diBrdPerSlt);
	p_ProdRcpCurrRcp3McMod			:= ADR(a_tyCurrRcp[3].usiMcMod);
	p_ProdRcpCurrRcp3TopToBtm		:= ADR(a_tyCurrRcp[3].bTopToBtm);
	p_ProdRcpCurrRcp3GapBtwnBrd		:= ADR(a_tyCurrRcp[3].bGapBwtnBrd);
	p_ProdRcpCurrRcp3LongBrd		:= ADR(a_tyCurrRcp[3].bLongBrd);
	p_ProdRcpCurrRcp3MinReqFreeBffr	:= ADR(a_tyCurrRcp[3].diMinReqFreeBffr);
	p_ProdRcpCurrRcp3DisplayInfo	:= ADR(a_tyCurrRcp[3].sDisplayInfo);
	p_ProdRcpCurrRcp3LastModified	:= ADR(a_tyCurrRcp[3].dtLastModified);
	p_ProdRcpCurrRcp3Width2 		:= ADR(a_tyCurrRcp[3].diWidthInUM2);
	p_ProdRcpCurrRcp3PshrPulerOffset:= ADR(a_tyCurrRcp[3].diPshrOffset);
	p_ProdRcpCurrRcp3MtrPshrExtSpd	:= ADR(a_tyCurrRcp[3].diMtrPshrExtSpd);
	p_ProdRcpCurrRcp3MtrPshrExtTorq	:= ADR(a_tyCurrRcp[3].diMtrPshrExtTorq);
	p_ProdRcpCurrRcp3PshrOffset		:= ADR(a_tyCurrRcp[3].diPshrOffset);

	p_ProdRcpCurrRcp4				:= ADR(a_tyCurrRcp[4]);
	p_ProdRcpCurrRcp4Nm				:= ADR(a_tyCurrRcp[4].sRcpNm);
	p_ProdRcpCurrRcp4Width			:= ADR(a_tyCurrRcp[4].diWidthInUM);
	p_ProdRcpCurrRcp4MinSltValue	:= ADR(a_tyCurrRcp[4].diMinSltValue);
	p_ProdRcpCurrRcp4MaxSltValue	:= ADR(a_tyCurrRcp[4].diMaxSltValue);
	p_ProdRcpCurrRcp4Pitch			:= ADR(a_tyCurrRcp[4].diPitch);
	p_ProdRcpCurrRcp4BrdPerSlt		:= ADR(a_tyCurrRcp[4].diBrdPerSlt);
	p_ProdRcpCurrRcp4McMod			:= ADR(a_tyCurrRcp[4].usiMcMod);
	p_ProdRcpCurrRcp4TopToBtm		:= ADR(a_tyCurrRcp[4].bTopToBtm);
	p_ProdRcpCurrRcp4GapBtwnBrd		:= ADR(a_tyCurrRcp[4].bGapBwtnBrd);
	p_ProdRcpCurrRcp4LongBrd		:= ADR(a_tyCurrRcp[4].bLongBrd);
	p_ProdRcpCurrRcp4MinReqFreeBffr	:= ADR(a_tyCurrRcp[4].diMinReqFreeBffr);
	p_ProdRcpCurrRcp4DisplayInfo	:= ADR(a_tyCurrRcp[4].sDisplayInfo);
	p_ProdRcpCurrRcp4LastModified	:= ADR(a_tyCurrRcp[4].dtLastModified);
	p_ProdRcpCurrRcp4Width2 		:= ADR(a_tyCurrRcp[4].diWidthInUM2);
	p_ProdRcpCurrRcp4PshrPulerOffset:= ADR(a_tyCurrRcp[4].diPshrOffset);
	p_ProdRcpCurrRcp4MtrPshrExtSpd	:= ADR(a_tyCurrRcp[4].diMtrPshrExtSpd);
	p_ProdRcpCurrRcp4MtrPshrExtTorq	:= ADR(a_tyCurrRcp[4].diMtrPshrExtTorq);
	p_ProdRcpCurrRcp4PshrOffset		:= ADR(a_tyCurrRcp[4].diPshrOffset);

	p_ProdRcpCurrRcp5				:= ADR(a_tyCurrRcp[5]);
	p_ProdRcpCurrRcp5Nm				:= ADR(a_tyCurrRcp[5].sRcpNm);
	p_ProdRcpCurrRcp5Width			:= ADR(a_tyCurrRcp[5].diWidthInUM);
	p_ProdRcpCurrRcp5MinSltValue	:= ADR(a_tyCurrRcp[5].diMinSltValue);
	p_ProdRcpCurrRcp5MaxSltValue	:= ADR(a_tyCurrRcp[5].diMaxSltValue);
	p_ProdRcpCurrRcp5Pitch			:= ADR(a_tyCurrRcp[5].diPitch);
	p_ProdRcpCurrRcp5BrdPerSlt		:= ADR(a_tyCurrRcp[5].diBrdPerSlt);
	p_ProdRcpCurrRcp5McMod			:= ADR(a_tyCurrRcp[5].usiMcMod);
	p_ProdRcpCurrRcp5TopToBtm		:= ADR(a_tyCurrRcp[5].bTopToBtm);
	p_ProdRcpCurrRcp5GapBtwnBrd		:= ADR(a_tyCurrRcp[5].bGapBwtnBrd);
	p_ProdRcpCurrRcp5LongBrd		:= ADR(a_tyCurrRcp[5].bLongBrd);
	p_ProdRcpCurrRcp5MinReqFreeBffr	:= ADR(a_tyCurrRcp[5].diMinReqFreeBffr);
	p_ProdRcpCurrRcp5DisplayInfo	:= ADR(a_tyCurrRcp[5].sDisplayInfo);
	p_ProdRcpCurrRcp5LastModified	:= ADR(a_tyCurrRcp[5].dtLastModified);
	p_ProdRcpCurrRcp5Width2			:= ADR(a_tyCurrRcp[5].diWidthInUM2);
	p_ProdRcpCurrRcp5PshrPulerOffset:= ADR(a_tyCurrRcp[5].diPshrOffset);
	p_ProdRcpCurrRcp5MtrPshrExtSpd	:= ADR(a_tyCurrRcp[5].diMtrPshrExtSpd);
	p_ProdRcpCurrRcp5MtrPshrExtTorq	:= ADR(a_tyCurrRcp[5].diMtrPshrExtTorq);
	p_ProdRcpCurrRcp5PshrOffset		:= ADR(a_tyCurrRcp[5].diPshrOffset);

	(* Always Change If Project Change *)

END_PROGRAM
```

#### Act_InputConfig.st - Change By Project
```iecst
(** 2020-06-08 **)
ACTION Act_InitGlobal:

	(* Always Change If Project Change *)
	p_eLinkLCSMngRcpProdRcpAct ACCESS p_LCSMngRcpProdRcpAct;
	p_eLinkUIProdRcpAct ACCESS p_UIProdRcpAct;
	p_tyInfoIn ACCESS p_UIProdRcpInfoIn;
	p_tyCurrRcpWr ACCESS p_UIProdRcpCurrRcpWr;

	//Input to Process
	tylocalProdRcp.In.udiRstErr 		:= g_tyRstErrOut.udiRstErr;
	tylocalProdRcp.In.sSearch			:= g_tyUIOut.sProdRcpSearch;
	tylocalProdRcp.In.sScan				:= g_tyUIOut.sProdRcpScan;
	tylocalProdRcp.In.sProgNm			:= g_tyNtParamCurr.sProdRcpProgNm;
	tylocalProdRcp.In.bWidth2Prep		:= g_tyNtParamCurr.bLFProdWidth2Prep;

	(* Always Change If Project Change *)

	IF g_tyStartUp.bRun THEN
		p_eAct ACCESS p_StartupProdRcpAct;
	ELSE
		IF tylocalProdRcp.Out.eStatus = Idle THEN
			IF g_tyNtParamCurr.bLCSManageRcpPrep AND g_tyMcParamCurr.bLCSManageRcpEn THEN
				IF p_eLinkLCSMngRcpProdRcpAct <> ProdRcpActIdle THEN
					p_eAct ACCESS p_LCSMngRcpProdRcpAct;
					p_tyInfoIn ACCESS p_LCSMngRcpProdRcpInfoIn;
				ELSIF p_eLinkUIProdRcpAct <> ProdRcpActIdle THEN
					p_eAct ACCESS p_UIProdRcpAct;
					p_tyInfoIn ACCESS p_UIProdRcpInfoIn;

					p_tyInfoIn.dtLastModified	:= g_tyTime.dtCurrDT;
				END_IF
			ELSE
				p_eAct ACCESS p_UIProdRcpAct;
				p_tyInfoIn ACCESS p_UIProdRcpInfoIn;
				p_tyInfoIn.dtLastModified	:= g_tyTime.dtCurrDT;
			END_IF
		END_IF
	END_IF

	IF (p_eAct = ProdRcpActAddEdit) OR (p_eAct = ProdRcpActAdd) OR (p_eAct = ProdRcpActEdit) THEN

		rWidthInMM				:= DINT_TO_REAL(p_tyInfoIn.diWidthInUM);
		rWidthInMM2				:= DINT_TO_REAL(p_tyInfoIn.diWidthInUM2);
		rWidthInMM				:= rWidthInMM / 1000;
		rWidthInMM2				:= rWidthInMM2 / 1000;
		sWidthInMM				:= REAL_TO_STRING(rWidthInMM);
		sWidthInMM2				:= REAL_TO_STRING(rWidthInMM2);

		IF tylocalProdRcp.In.bWidth2Prep THEN
			p_tyInfoIn.sDisplayInfo	:= sWidthInMM;
			p_tyInfoIn.sDisplayInfo	:= CONCAT(p_tyInfoIn.sDisplayInfo , ' | ');
			p_tyInfoIn.sDisplayInfo	:= CONCAT(p_tyInfoIn.sDisplayInfo , sWidthInMM2);
			p_tyInfoIn.sDisplayInfo	:= CONCAT(p_tyInfoIn.sDisplayInfo , ' mm');
		ELSE
			p_tyInfoIn.sDisplayInfo	:= sWidthInMM;
			p_tyInfoIn.sDisplayInfo	:= CONCAT(p_tyInfoIn.sDisplayInfo , ' mm');
		END_IF
	END_IF

END_ACTION
```

#### Act_OutputConfig.st - Change By Project
```iecst
ACTION Act_OutputConfig:

  g_tyProdRcp := tylocalProdRcp.Out;

END_ACTION
```

#### Cyclic.st - Do Not Change!!!
```iecst
(** 2019-03-29 **)
PROGRAM _CYCLIC

	IF bInitialDone = FALSE THEN
		F g_tyStartUp.bNtSettingsLoadDone = TRUE THEN
			bInitialDone	:= TRUE;

			Act_Initial;
		END_IF

	ELSE

		Act_InputConfig;
		Act_Main;
		Act_OutputConfig;
		Act_Alarm;

	END_IF

END_PROGRAM
```

#### Act_InitLocal.st - Do Not Change!!!
```iecst
(** 2020-06-08 **)
ACTION Act_InitLocal:

	//Input Reference Link To Local Variable
	p_eAct ACCESS ADR(eAct);
	p_udiMax ACCESS ADR(c_udiProdRcpMax);
	p_udiRstErr ACCESS ADR(udiRstErr);
	p_dtCurrDT ACCESS ADR(dtCurrDT);
	p_sSearch ACCESS ADR(sSearch);
	p_sScan ACCESS ADR(sScan);
	p_tyInfoIn ACCESS ADR(tyInfoIn);
	p_tyCurrRcpWr ACCESS ADR(tyCurrRcpWr);
	p_sListFileName ACCESS ADR(sListFileName);
	p_sSingleFileName ACCESS ADR(sSingleFileName);
	p_sProgNm ACCESS ADR(sProgNm);
	p_bNtSettingsLoadDone ACCESS ADR(bNtSettingsLoadDone);
	p_bWidth2Prep ACCESS ADR(bWidth2Prep);
	p_uiSortNo ACCESS ADR(uiSortNo);
END_ACTION
```

#### Act_Initial.st - Do Not Change!!!
```iecst
(** 2019-06-10 **)
ACTION Act_Initial:

	//Initial
	sStatTxt	:= a_sStatText[tylocalProdRcp.Out.eStat];

	//Initial Addressing
	p_eAct ACCESS ADR (eAct);
	p_tyInfoIn ACCESS ADR(tyInfoIn);
	p_tyCurrRcpWr ACCESS ADR(tyCurrRcpWr);
	p_udiMax ACCESS ADR(c_udiProdRcpMax);

	fbDirCreate1.sDevice	:= 'C';
	fbDirCreate1.sDirName	:= 'User';
	fbDirCreate1(bEn := FALSE);

	fbDirCreate2.sDevice	:= 'User';
	fbDirCreate2.sDirName	:= 'ProductRecipe';
	fbDirCreate2(bEn := FALSE);

	fbFileReadList.sDevice		:= 'ProdRcp';
	fbFileReadList.sFile		:= g_tyNtParamCurr.sProdRcpListFileNm;
	fbFileReadList.udiOffset	:= 0;
	fbFileReadList.p_Dest		:= ADR(a_tyCurrList);
	fbFileReadList.udiLen		:= SIZEOF(a_tyCurrList);
	fbFileReadList(bEn := FALSE);

	fbFileWriteList.sDevice		:= 'ProdRcp';
	fbFileWriteList.sFile		:= g_tyNtParamCurr.sProdRcpListFileNm;
	fbFileWriteList.udiOffset	:= 0;
	fbFileWriteList.p_Src		:= ADR(a_tyListTemp);
	fbFileWriteList.udiLen		:= SIZEOF(a_tyListTemp);
	fbFileWriteList.udiOption	:= 0;
	fbFileWriteList(bEn := FALSE);

	fbFileReadSingle.sDevice	:= 'ProdRcp';
	fbFileReadSingle.sFile		:= g_tyNtParamCurr.sProdRcpSingleFileNm;
	fbFileReadSingle.udiOffset	:= 0;
	fbFileReadSingle.p_Dest		:= ADR(a_tyCurrRcp[0]);
	fbFileReadSingle.udiLen		:= SIZEOF(a_tyCurrRcp[0]);
	fbFileReadSingle(bEn := FALSE);

	fbFileLoadSingle.sDevice	:= 'ProdRcp';
	fbFileLoadSingle.sFile		:= g_tyNtParamCurr.sProdRcpSingleFileNm;
	fbFileLoadSingle.udiOffset	:= 0;
	fbFileLoadSingle.p_Src		:= ADR(a_tyCurrRcp[0]);
	fbFileLoadSingle.udiLen		:= SIZEOF(a_tyCurrRcp[0]);
	fbFileLoadSingle.udiOption	:= 0;
	fbFileLoadSingle(bEn := FALSE);

	fbFileWriteSingle.sDevice	:= 'ProdRcp';
	fbFileWriteSingle.sFile		:= g_tyNtParamCurr.sProdRcpSingleFileNm;
	fbFileWriteSingle.udiOffset	:= 0;
	fbFileWriteSingle.p_Src		:= ADR(p_tyCurrRcpWr);
	fbFileWriteSingle.udiLen	:= SIZEOF(p_tyCurrRcpWr);
	fbFileWriteSingle.udiOption	:= 0;
	fbFileWriteSingle(bEn := FALSE);

END_ACTION
```

#### Act_Main.st - Do Not Change!!!
```iecst
ACTION Act_Main:

	//Set p_eAct
	IF tylocalProdRcp.Out.eStatus = Idle THEN
		tylocalProdRcp.Out.eStat	:= p_eAct;
	END_IF

	//Main
	CASE tylocalProdRcp.Out.eStat OF

		ProdRcpActIdle:
			IF tylocalProdRcp.Out.eStatus <> Idle THEN	//Reset Data
				//Private
				fbDirCreate1(bEn := FALSE);
				fbDirCreate2(bEn := FALSE);
				fbFileReadList(bEn := FALSE);
				fbFileWriteList(bEn := FALSE);
				fbFileReadSingle(bEn := FALSE);
				fbFileWriteSingle(bEn := FALSE);
				fbFileLoadSingle(bEn := FALSE);
				usiStep				:= 0;
				udiAddStatus		:= 0;

				bNmExist		:= FALSE;
				bNmNotExist		:= FALSE;
				bNmEmpty		:= FALSE;
				bListFull		:= FALSE;
				bFileNotFound	:= FALSE;
				iTotalRcp 		:= 0;

				memset(ADR(tyTempRecipe), 0 , SIZEOF(tyTempRecipe));

				tylocalProdRcp.Out.sStatTxt	:= a_sStatText[tylocalProdRcp.Out.eStat];

			END_IF

			tylocalProdRcp.Out.eStatus	:= Idle;

		ProdRcpActCreateDir:
			IF tylocalProdRcp.Out.eStatus = Idle OR tylocalProdRcp.Out.eStatus = Busy THEN

				tylocalProdRcp.Out.eStatus	:= Busy;

				tylocalProdRcp.Out.sStatTxt	:= a_sStatText[tylocalProdRcp.Out.eStat];

				CASE usiStep OF
					0:
						fbDirCreate1(bEn := TRUE);
						IF fbDirCreate1.udiStatus = 0 THEN
							usiStep	:= 1;
						ELSIF fbDirCreate1.udiStatus < 65534 THEN
							tylocalProdRcp.Out.eStatus		:= Error;

							IF fbDirCreate1.udiStatus = 1908 THEN
								udiStatus	:= 10000;	//Create User Directory Error
							ELSE
								udiStatus	:= fbDirCreate1.udiStatus;
							END_IF
						END_IF

					1:
						fbDirCreate2(bEn := TRUE);
						IF fbDirCreate2.udiStatus = 0 THEN
							tylocalProdRcp.Out.eStatus	:= Done;
						ELSIF fbDirCreate2.udiStatus < 65534 THEN
							tylocalProdRcp.Out.eStatus		:= Error;

							IF fbDirCreate2.udiStatus = 1908 THEN
								udiStatus	:= 10001;	//Create Product Recipe Directory Error
							ELSE
								udiStatus	:= fbDirCreate2.udiStatus;
							END_IF
						END_IF

				END_CASE

			END_IF

		ProdRcpActAddEdit:
			IF tylocalProdRcp.Out.eStatus = Idle OR tylocalProdRcp.Out.eStatus = Busy THEN

				tylocalProdRcp.Out.eStatus	:= Busy;

				tylocalProdRcp.Out.sStatTxt	:= a_sStatText[tylocalProdRcp.Out.eStat];

				CASE usiStep OF
					0:	//Edit Recipe
						udiAddStatus	:= fRecipeAddEdit(ADR(p_tyInfoIn) , ADR(a_tyListTemp) , SIZEOF(a_tyListTemp[1]) , ADR(a_tyListTemp[1].sRcpNm) , SIZEOF(a_tyListTemp[1].sRcpNm) , p_udiMax);

						IF udiAddStatus = 1600 THEN	//Recipe Name Empty
							bNmEmpty	:= TRUE;
							tylocalProdRcp.Out.eStatus		:= Done;

						ELSIF udiAddStatus = 1601 THEN	//Recipe Full
							bListFull	:= TRUE;
							tylocalProdRcp.Out.eStatus		:= Done;

						ELSIF udiAddStatus = 0 THEN	//OK
							usiStep	:= 1;

						END_IF

					1:	//Write Into File
						fbFileWriteList(bEn := TRUE);

						IF fbFileWriteList.udiStatus = 0 THEN
							a_tyCurrList						:= a_tyListTemp;
							tylocalProdRcp.Out.eStatus			:= Done;

						ELSIF fbFileWriteList.udiStatus < 65534 THEN
							a_tyListTemp	:= a_tyCurrList;
							tylocalProdRcp.Out.eStatus			:= Error;

							IF fbFileWriteList.udiStatus = 1900 THEN
								udiStatus	:= 10002;	//File Open Error While Adding & Editing
							ELSIF fbFileWriteList.udiStatus = 1901 THEN
								udiStatus	:= 10003;	//File Create Error While Adding & Editing
							ELSIF fbFileWriteList.udiStatus = 1903 THEN
								udiStatus	:= 10004;	//File Write Error While Adding & Editing
							ELSIF fbFileWriteList.udiStatus = 1904 THEN
								udiStatus	:= 10005;	//File Close Error While Adding & Editing
							ELSIF fbFileWriteList.udiStatus = 1914 THEN
								udiStatus	:= 10013;	//Directory Does Not Exist While Adding & Editing
							ELSE
								udiStatus	:= fbFileWriteList.udiStatus;
							END_IF
						END_IF

				END_CASE

			END_IF

		ProdRcpActDel:
			IF tylocalProdRcp.Out.eStatus = Idle OR tylocalProdRcp.Out.eStatus = Busy THEN

				tylocalProdRcp.Out.eStatus	:= Busy;

				tylocalProdRcp.Out.sStatTxt	:= a_sStatText[tylocalProdRcp.Out.eStat];

				CASE usiStep OF
					0:	//Edit User
						udiAddStatus	:= fRecipeDelete(ADR(p_tyInfoIn) , ADR(a_tyListTemp) , SIZEOF(a_tyListTemp[1]) , ADR(a_tyListTemp[1].sRcpNm) , SIZEOF(a_tyListTemp[1].sRcpNm) , p_udiMax);

						IF udiAddStatus = 1600 THEN	//Recipe Name Empty
							bNmEmpty	:= TRUE;
							tylocalProdRcp.Out.eStatus		:= Done;

						ELSIF udiAddStatus = 1603 THEN	//Recipe Not Exist
							bNmNotExist	:= TRUE;
							tylocalProdRcp.Out.eStatus		:= Done;

						ELSIF udiAddStatus = 0 THEN	//OK
							usiStep	:= 1;

						END_IF

					1:	//Write Into File
						fbFileWriteList(bEn := TRUE);

						IF fbFileWriteList.udiStatus = 0 THEN
							a_tyCurrList	:= a_tyListTemp;
							tylocalProdRcp.Out.eStatus			:= Done;

						ELSIF fbFileWriteList.udiStatus < 65534 THEN
							a_tyListTemp	:= a_tyCurrList;
							tylocalProdRcp.Out.eStatus			:= Error;

							IF fbFileWriteList.udiStatus = 1900 THEN
								udiStatus	:= 10006;	//File Open Error While Deleting
							ELSIF fbFileWriteList.udiStatus = 1901 THEN
								udiStatus	:= 10007;	//File Create Error While Deleting
							ELSIF fbFileWriteList.udiStatus = 1903 THEN
								udiStatus	:= 10008;	//File Write Error While Deleting
							ELSIF fbFileWriteList.udiStatus = 1904 THEN
								udiStatus	:= 10009;	//File Close Error While Deleting
							ELSIF fbFileWriteList.udiStatus = 1914 THEN
								udiStatus	:= 10014;	//Directory Does Not Exist While Deleting
							ELSE
								udiStatus	:= fbFileWriteList.udiStatus;
							END_IF

						END_IF

				END_CASE

			END_IF

		ProdRcpActGetInfo:
			IF tylocalProdRcp.Out.eStatus = Idle OR tylocalProdRcp.Out.eStatus = Busy THEN

				tylocalProdRcp.Out.sStatTxt	:= a_sStatText[tylocalProdRcp.Out.eStat];

				IF p_tyInfoIn.sRcpNm = '' THEN
					bNmEmpty	:= TRUE;
					bNmNotExist	:= TRUE;
				ELSE
					bNmNotExist	:= (fRecipeGetInfo(p_tyInfoIn.sRcpNm , ADR(tyInfoOut) , ADR(a_tyCurrList) , SIZEOF(a_tyCurrList[1]) , ADR(a_tyCurrList[1].sRcpNm) , SIZEOF(a_tyCurrList[1].sRcpNm) , p_udiMax)) = 0;
				END_IF

				tylocalProdRcp.Out.eStatus	:= Done;

			END_IF

		ProdRcpActGetList:
			IF tylocalProdRcp.Out.eStatus = Idle OR tylocalProdRcp.Out.eStatus = Busy THEN

				tylocalProdRcp.Out.eStatus	:= Busy;

				tylocalProdRcp.Out.sStatTxt	:= a_sStatText[tylocalProdRcp.Out.eStat];

				fbFileReadList(bEn := TRUE);

				IF fbFileReadList.udiStatus = 0 THEN
					a_tyListTemp	:= a_tyCurrList;
					tylocalProdRcp.Out.eStatus			:= Done;

				ELSIF fbFileReadList.udiStatus < 65534 THEN
					tylocalProdRcp.Out.eStatus		:= Error;

					IF fbFileReadList.udiStatus = 1900 THEN
						udiStatus	:= 10010;	//File Open Error While Getting List
					ELSIF fbFileReadList.udiStatus = 1902 THEN
						udiStatus	:= 10011;	//File Read Error While Getting List
					ELSIF fbFileReadList.udiStatus = 1904 THEN
						udiStatus	:= 10012;	//File Close Error While Getting List
					ELSIF fbFileReadList.udiStatus = 1915 THEN
						tylocalProdRcp.Out.eStatus			:= Done;
						bFileNotFound	:= TRUE;
					ELSE
						udiStatus	:= fbFileReadList.udiStatus;
					END_IF

				END_IF

			END_IF

		ProdRcpActFilter:

			IF tylocalProdRcp.Out.eStatus = Idle OR tylocalProdRcp.Out.eStatus = Busy THEN

				tylocalProdRcp.Out.eStatus := Busy;

				sStatTxt	:= a_sStatText[tylocalProdRcp.Out.eStat];

				CASE usiStep OF
					0:
						fRecipeFilter(tylocalProdRcp.In.sSearch , ADR(a_tyFilterList) , ADR(a_tyCurrList) , SIZEOF(a_tyCurrList[1]) , ADR(a_tyCurrList[1].sRcpNm) ,
						SIZEOF(a_tyCurrList[1].sRcpNm) , p_udiMax, 0, 499, iFilterCtr);
						usiStep := 1;
					1:
						fRecipeFilter(tylocalProdRcp.In.sSearch , ADR(a_tyFilterList) , ADR(a_tyCurrList) , SIZEOF(a_tyCurrList[1]) , ADR(a_tyCurrList[1].sRcpNm) ,
						SIZEOF(a_tyCurrList[1].sRcpNm) , p_udiMax, 500, 999, iFilterCtr);
						usiStep := 2;
					2:
						fRecipeFilter(tylocalProdRcp.In.sSearch , ADR(a_tyFilterList) , ADR(a_tyCurrList) , SIZEOF(a_tyCurrList[1]) , ADR(a_tyCurrList[1].sRcpNm) ,
						SIZEOF(a_tyCurrList[1].sRcpNm) , p_udiMax, 1000, 1499, iFilterCtr);
						usiStep := 3;
					3:
						fRecipeFilter(tylocalProdRcp.In.sSearch , ADR(a_tyFilterList) , ADR(a_tyCurrList) , SIZEOF(a_tyCurrList[1]) , ADR(a_tyCurrList[1].sRcpNm) ,
						SIZEOF(a_tyCurrList[1].sRcpNm) , p_udiMax, 1500, 1999, iFilterCtr);
						tylocalProdRcp.Out.eStatus := Done;

				END_CASE

			END_IF
		ProdRcpActLoadRcp:
			IF tylocalProdRcp.Out.eStatus = Idle OR tylocalProdRcp.Out.eStatus = Busy THEN

				tylocalProdRcp.Out.sStatTxt	:= a_sStatText[tylocalProdRcp.Out.eStat];

				CASE usiStep OF
					0:	//Get Current Recipe
						IF p_tyInfoIn.sRcpNm = '' THEN
							bNmEmpty	:= TRUE;
							bNmNotExist	:= TRUE;

							tylocalProdRcp.Out.eStatus	:= Done;
						ELSE
							bNmNotExist	:= (fRecipeGetInfo(p_tyInfoIn.sRcpNm , ADR(a_tyCurrRcp[0]) , ADR(a_tyCurrList) , SIZEOF(a_tyCurrList[1]) , ADR(a_tyCurrList[1].sRcpNm) , SIZEOF(a_tyCurrList[1].sRcpNm) , p_udiMax)) = 0;

							IF bNmNotExist = TRUE THEN
								tylocalProdRcp.Out.eStatus	:= Done;
							ELSE
								usiStep	:= 1;
							END_IF

						END_IF

					1:	//Write Into File
						fbFileLoadSingle(bEn := TRUE);

						IF fbFileLoadSingle.udiStatus = 0 THEN
							tylocalProdRcp.Out.eStatus			:= Done;
						ELSIF fbFileLoadSingle.udiStatus < 65534 THEN
							tylocalProdRcp.Out.eStatus			:= Error;

							IF fbFileLoadSingle.udiStatus = 1900 THEN
								udiStatus	:= 10025;	//File Open Error While Loading Current Recipe
							ELSIF fbFileLoadSingle.udiStatus = 1901 THEN
								udiStatus	:= 10026;	//File Create Error While Loading Current Recipe
							ELSIF fbFileLoadSingle.udiStatus = 1903 THEN
								udiStatus	:= 10027;	//File Write Error While Loading Current Recipe
							ELSIF fbFileLoadSingle.udiStatus = 1904 THEN
								udiStatus	:= 10028;	//File Close Error While Loading Current Recipe
							ELSIF fbFileLoadSingle.udiStatus = 1914 THEN
								udiStatus	:= 10029;	//Directory Does Not Exist While Loading Current Recipe
							ELSE
								udiStatus	:= fbFileLoadSingle.udiStatus;
							END_IF
						END_IF

				END_CASE

			END_IF

		ProdRcpActAdd:
			IF tylocalProdRcp.Out.eStatus = Idle OR tylocalProdRcp.Out.eStatus = Busy THEN

				tylocalProdRcp.Out.eStatus	:= Busy;

				tylocalProdRcp.Out.sStatTxt	:= a_sStatText[tylocalProdRcp.Out.eStat];

				CASE usiStep OF
					0:	//Edit Recipe
						udiAddStatus	:= fRecipeAdd(ADR(p_tyInfoIn) , ADR(a_tyListTemp) , SIZEOF(a_tyListTemp[1]) , ADR(a_tyListTemp[1].sRcpNm) , SIZEOF(a_tyListTemp[1].sRcpNm) , p_udiMax);

						IF udiAddStatus = 1600 THEN	//Recipe Name Empty
							bNmEmpty	:= TRUE;
							tylocalProdRcp.Out.eStatus		:= Done;

						ELSIF udiAddStatus = 1601 THEN	//Recipe Full
							bListFull	:= TRUE;
							tylocalProdRcp.Out.eStatus		:= Done;

						ELSIF udiAddStatus = 1602 THEN	//Recipe Name Exist
							bNmExist	:= TRUE;
							tylocalProdRcp.Out.eStatus		:= Done;

						ELSIF udiAddStatus = 0 THEN	//OK
							usiStep	:= 1;

						END_IF

					1:	//Write Into File
						fbFileWriteList(bEn := TRUE);

						IF fbFileWriteList.udiStatus = 0 THEN
							a_tyCurrList	:= a_tyListTemp;
							tylocalProdRcp.Out.eStatus			:= Done;

						ELSIF fbFileWriteList.udiStatus < 65534 THEN
							a_tyListTemp	:= a_tyCurrList;
							tylocalProdRcp.Out.eStatus			:= Error;

							IF fbFileWriteList.udiStatus = 1900 THEN
								udiStatus	:= 10015;	//File Open Error While Adding
							ELSIF fbFileWriteList.udiStatus = 1901 THEN
								udiStatus	:= 10016;	//File Create Error While Adding
							ELSIF fbFileWriteList.udiStatus = 1903 THEN
								udiStatus	:= 10017;	//File Write Error While Adding
							ELSIF fbFileWriteList.udiStatus = 1904 THEN
								udiStatus	:= 10018;	//File Close Error While Adding
							ELSIF fbFileWriteList.udiStatus = 1914 THEN
								udiStatus	:= 10019;	//Directory Does Not Exist While Adding
							ELSE
								udiStatus	:= fbFileWriteList.udiStatus;
							END_IF
						END_IF
				END_CASE

			END_IF

		ProdRcpActEdit:
			IF tylocalProdRcp.Out.eStatus = Idle OR tylocalProdRcp.Out.eStatus = Busy THEN

				tylocalProdRcp.Out.eStatus	:= Busy;

				tylocalProdRcp.Out.sStatTxt	:= a_sStatText[tylocalProdRcp.Out.eStat];

				CASE usiStep OF
					0:	//Edit Recipe
						udiAddStatus	:= fRecipeEdit(ADR(p_tyInfoIn) , ADR(a_tyListTemp) , SIZEOF(a_tyListTemp[1]) , ADR(a_tyListTemp[1].sRcpNm) , SIZEOF(a_tyListTemp[1].sRcpNm) , p_udiMax);

						IF udiAddStatus = 1600 THEN	//Recipe Name Empty
							bNmEmpty	:= TRUE;
							tylocalProdRcp.Out.eStatus		:= Done;

						ELSIF udiAddStatus = 1603 THEN	//Recipe Not Exist
							bNmNotExist	:= TRUE;
							tylocalProdRcp.Out.eStatus		:= Done;

						ELSIF udiAddStatus = 0 THEN	//OK
							usiStep	:= 1;

						END_IF

					1:	//Write Into File
						fbFileWriteList(bEn := TRUE);

						IF fbFileWriteList.udiStatus = 0 THEN
							a_tyCurrList	:= a_tyListTemp;
							tylocalProdRcp.Out.eStatus			:= Done;

						ELSIF fbFileWriteList.udiStatus < 65534 THEN
							a_tyListTemp	:= a_tyCurrList;
							tylocalProdRcp.Out.eStatus			:= Error;

							IF fbFileWriteList.udiStatus = 1900 THEN
								udiStatus	:= 10020;	//File Open Error While Adding & Editing
							ELSIF fbFileWriteList.udiStatus = 1901 THEN
								udiStatus	:= 10021;	//File Create Error While Adding & Editing
							ELSIF fbFileWriteList.udiStatus = 1903 THEN
								udiStatus	:= 10022;	//File Write Error While Adding & Editing
							ELSIF fbFileWriteList.udiStatus = 1904 THEN
								udiStatus	:= 10023;	//File Close Error While Adding & Editing
							ELSIF fbFileWriteList.udiStatus = 1914 THEN
								udiStatus	:= 10024;	//Directory Does Not Exist While Adding & Editing
							ELSE
								udiStatus	:= fbFileWriteList.udiStatus;
							END_IF
						END_IF

				END_CASE

			END_IF

		ProdRcpActReadCurrRcp:
			IF tylocalProdRcp.Out.eStatus = Idle OR tylocalProdRcp.Out.eStatus = Busy THEN

				tylocalProdRcp.Out.eStatus	:= Busy;

				tylocalProdRcp.Out.sStatTxt	:= a_sStatText[tylocalProdRcp.Out.eStat];

				fbFileReadSingle(bEn := TRUE);
				IF fbFileReadSingle.udiStatus = 0 THEN
					tylocalProdRcp.Out.eStatus			:= Done;

				ELSIF fbFileReadSingle.udiStatus < 65534 THEN
					tylocalProdRcp.Out.eStatus		:= Error;

					IF fbFileReadSingle.udiStatus = 1900 THEN
						udiStatus	:= 10030;	//File Open Error While Reading Current Recipe
					ELSIF fbFileReadSingle.udiStatus = 1902 THEN
						udiStatus	:= 10031;	//File Read Error While Reading Current Recipe
					ELSIF fbFileReadSingle.udiStatus = 1904 THEN
						udiStatus	:= 10032;	//File Close Error While Reading Current Recipe
					ELSIF fbFileReadSingle.udiStatus = 1915 THEN
						tylocalProdRcp.Out.eStatus			:= Done;
						bFileNotFound	:= TRUE;
					ELSE
						udiStatus	:= fbFileReadSingle.udiStatus;
					END_IF
				END_IF

			END_IF

		ProdRcpActWriteCurrRcpParam:
			IF tylocalProdRcp.Out.eStatus = Idle OR tylocalProdRcp.Out.eStatus = Busy THEN

				tylocalProdRcp.Out.sStatTxt	:= a_sStatText[tylocalProdRcp.Out.eStat];

				fbFileWriteSingle(bEn := TRUE);

				IF fbFileWriteSingle.udiStatus = 0 THEN
					a_tyCurrRcp[0]	:= p_tyCurrRcpWr;
					tylocalProdRcp.Out.eStatus			:= Done;
				ELSIF fbFileWriteSingle.udiStatus < 65534 THEN
					tylocalProdRcp.Out.eStatus			:= Error;

					IF fbFileWriteSingle.udiStatus = 1900 THEN
						udiStatus	:= 10033;	//File Open Error While Writing Current Recipe Parameter
					ELSIF fbFileWriteSingle.udiStatus = 1901 THEN
						udiStatus	:= 10034;	//File Create Error While Writing Current Recipe Parameter
					ELSIF fbFileWriteSingle.udiStatus = 1903 THEN
						udiStatus	:= 10035;	//File Write Error While Writing Current Recipe Parameter
					ELSIF fbFileWriteSingle.udiStatus = 1904 THEN
						udiStatus	:= 10036;	//File Close Error While Writing Current Recipe Parameter
					ELSIF fbFileWriteSingle.udiStatus = 1914 THEN
						udiStatus	:= 10037;	//Directory Does Not Exist Writing Current Recipe Parameter
					ELSE
						udiStatus	:= fbFileWriteSingle.udiStatus;
					END_IF
				END_IF

			END_IF

		ProdRcpActSaveList:
			IF tylocalProdRcp.Out.eStatus = Idle OR tylocalProdRcp.Out.eStatus = Busy THEN

				tylocalProdRcp.Out.eStatus	:= Busy;

				tylocalProdRcp.Out.sStatTxt	:= a_sStatText[tylocalProdRcp.Out.eStat];

				CASE usiStep OF

					0:
						a_tyListTemp	:= a_tyCurrList;

						fbFileWriteList(bEn := TRUE);

						IF fbFileWriteList.udiStatus = 0 THEN
							tylocalProdRcp.Out.eStatus			:= Done;

						ELSIF fbFileWriteList.udiStatus < 65534 THEN
							tylocalProdRcp.Out.eStatus			:= Error;

							IF fbFileWriteList.udiStatus = 1900 THEN
								udiStatus	:= 10038;	//File Open Error While Saving List
							ELSIF fbFileWriteList.udiStatus = 1901 THEN
								udiStatus	:= 10039;	//File Create Error While Saving List
							ELSIF fbFileWriteList.udiStatus = 1903 THEN
								udiStatus	:= 10040;	//File Write Error While Saving List
							ELSIF fbFileWriteList.udiStatus = 1904 THEN
								udiStatus	:= 10041;	//File Close Error While Saving List
							ELSIF fbFileWriteList.udiStatus = 1914 THEN
								udiStatus	:= 10042;	//Directory Does Not Exist While Saving List
							ELSE
								udiStatus	:= fbFileWriteList.udiStatus;
							END_IF
						END_IF

				END_CASE

			END_IF

		ProdRcpActSort:
			IF tylocalProdRcp.Out.eStatus = Idle OR tylocalProdRcp.Out.eStatus = Busy THEN

				tylocalProdRcp.Out.sStatTxt	:= a_sStatText[tylocalProdRcp.Out.eStat];

				CASE usiStep OF

					0:

						FOR udi := 1 TO c_udiProdRcpMax DO
							IF tylocalProdRcp.In.sSearch <> '' THEN
								IF a_tyFilterList[udi].sRcpNm = '' THEN
									usiStep := 1;
									EXIT;
								ELSIF udi = c_udiProdRcpMax THEN
									iTotalRcp := UDINT_TO_INT(c_udiProdRcpMax);
									usiStep := 1;
									EXIT;
								ELSE
									iTotalRcp := iTotalRcp +1;
								END_IF
							ELSE
								IF a_tyCurrList[udi].sRcpNm = '' THEN
									usiStep := 1;
									EXIT;
								ELSIF udi = c_udiProdRcpMax THEN
									iTotalRcp := UDINT_TO_INT(c_udiProdRcpMax);
									usiStep := 1;
									EXIT;
								ELSE
									iTotalRcp := iTotalRcp +1;
								END_IF
							END_IF
						END_FOR

					1:
						IF tylocalProdRcp.In.sSearch <> '' THEN
							memcpy(ADR(a_tySortList),ADR(a_tyFilterList), SIZEOF(a_tyFilterList));
						ELSE
							memcpy(ADR(a_tySortList),ADR(a_tyCurrList), SIZEOF(a_tyCurrList));
						END_IF

						iSortCurrentOuterCntr	:= 0;
						iSortCurrentInnerCntr	:= 1 ;

						udiSortCurrenTotalCntr	:= 0;

						usiStep := 2;

					2:

						IF iSortCurrentOuterCntr < iTotalRcp THEN

							FOR iSortCurrentInnerCntr:= iSortCurrentOuterCntr+1 TO iTotalRcp-1 DO

								IF fRecipeNmCompare(ADR(a_tySortList[iSortCurrentOuterCntr+1].sRcpNm),ADR(a_tySortList[iSortCurrentInnerCntr+1].sRcpNm),SIZEOF(a_tySortList[1].sRcpNm),ADR(sDebug)) THEN

									memcpy(ADR(tyTempRecipe), ADR(a_tySortList[iSortCurrentOuterCntr+1]), SIZEOF(a_tySortList[1]));
									memcpy(ADR(a_tySortList[iSortCurrentOuterCntr+1]), ADR(a_tySortList[iSortCurrentInnerCntr+1]), SIZEOF(a_tySortList[1]));
									memcpy(ADR(a_tySortList[iSortCurrentInnerCntr+1]), ADR(tyTempRecipe), SIZEOF(a_tySortList[1]));

								END_IF

								udiSortCurrenTotalCntr	:= udiSortCurrenTotalCntr + 1;

							END_FOR

							iSortCurrentOuterCntr	:= iSortCurrentOuterCntr + 1;

						ELSE
							usiStep := 3;
						END_IF

					3:
						tylocalProdRcp.Out.eStatus	:= Done;

				END_CASE

			END_IF

		ProdRcpActEndCharFilter:
			IF tylocalProdRcp.Out.eStatus = Idle OR tylocalProdRcp.Out.eStatus = Busy THEN

				tylocalProdRcp.Out.sStatTxt	:= a_sStatText[tylocalProdRcp.Out.eStat];

				fRecipeLastCharFilter(tylocalProdRcp.In.sScan , ADR(a_tyScanList) , ADR(a_tyCurrList) , SIZEOF(a_tyCurrList[1]) , ADR(a_tyCurrList[1].sRcpNm) , SIZEOF(a_tyCurrList[1].sRcpNm) , p_udiMax);

				tylocalProdRcp.Out.eStatus	:= Done;

			END_IF

	END_CASE

END_ACTION
```

#### Act_Alarm.st - Do Not Change!!!
```iecst
ACTION Act_Alarm:

	IF tylocalProdRcp.In.udiRstErr <> udiRstErrOld THEN
		bRstErr			:= TRUE;
		udiRstErrOld	:= tylocalProdRcp.In.udiRstErr;
	ELSE
		bRstErr			:= FALSE;
	END_IF

	//Reset Error
	IF (tylocalProdRcp.Out.eStatus = Error) AND bRstErr THEN
		p_eAct						:= ProdRcpActIdle;
		tylocalProdRcp.Out.eStat	:= ProdRcpActIdle;
	END_IF

	//Reset Done
	IF tylocalProdRcp.Out.eStatus = Done AND p_eAct = ProdRcpActIdle THEN
		tylocalProdRcp.Out.eStat	:= ProdRcpActIdle;
	END_IF

	//Error
	IF EDGEPOS(tylocalProdRcp.Out.eStatus = Error) THEN

		tylocalProdRcp.Out.tyAlmData.udiCode		:= udiStatus;
		tylocalProdRcp.Out.tyAlmData.eSeverity		:= AlmSeverityError;
		tylocalProdRcp.Out.tyAlmData.udiRunTime		:= tylocalProdRcp.Out.tyAlmData.udiRunTime + 1;
		tylocalProdRcp.Out.tyAlmData.bAlm			:= TRUE;
		tylocalProdRcp.Out.tyAlmData.udiModuleNum	:= udiModuleNum;
		g_tyAlmProgNm.sProdRcpProgNm				:= tylocalProdRcp.In.sProgNm;

	ELSIF bRstErr AND (tylocalProdRcp.Out.tyAlmData.udiCode <> 0) THEN

		tylocalProdRcp.Out.tyAlmData.udiCode	:= 0;
		tylocalProdRcp.Out.tyAlmData.eSeverity	:= AlmSeverityNA;
	    tylocalProdRcp.Out.tyAlmData.bAlm		:= FALSE;

		tylocalProdRcp.Out.sStatTxt	:= a_sStatText[tylocalProdRcp.Out.eStat];

	END_IF

END_ACTION
```

#### Local.var - Do Not Change!!!
```iecst
(*2020-07-24*)
(**)
VAR
	tylocalProdRcp : tyProdRcp;
	p_eAct : REFERENCE TO eProdRcpAction;
	p_udiMax : REFERENCE TO UDINT;
	p_tyInfoIn : REFERENCE TO tyProdRcpParam;
	p_tyCurrRcpWr : REFERENCE TO tyProdRcpParam;
	p_eLinkLCSMngRcpProdRcpAct : REFERENCE TO eProdRcpAction;
	p_eLinkUIProdRcpAct : REFERENCE TO eProdRcpAction;
	a_sStatText : ARRAY[0..50] OF STRING[200] := ['Idling','Creating Directory','Adding and Editing Files','Deleting Files','Get Info','Get List','Filtering Files','Loading Recipe','Adding Files','Editing Files','Reading Current Recipe','Writing Current Recipe Parameter','Saving Recipe List',38('')];
END_VAR
(**)
(*Local Alarm*)
VAR
	tyAlmData : tyAlmDat;
	a_tyAlmText : ARRAY[10000..10099] OF tyAlmTxt := [(sAlmText:='Create User Directory Error',sRcyText:='Unable To Create User Directory. Please Contact Nutek For A Possible Solution'),(sAlmText:='Create Product Recipe Directory Error',sRcyText:='Unable To Create Product Recipe Directory. Please Contact Nutek For A Possible Solution'),(sAlmText:='File Open Error While Adding & Editing',sRcyText:='An Error Was Encountered While Trying To Open File. Please Contact Nutek For A Possible Solution.'),(sAlmText:='File Create Error While Adding & Editing',sRcyText:='An Error Was Encountered While Trying To Create File. Please Contact Nutek For A Possible Solution.'),(sAlmText:='File Write Error While Adding & Editing',sRcyText:='An Error Was Encountered While Trying To Write File. Please Contact Nutek For A Possible Solution.'),(sAlmText:='File Close Error While Adding & Editing',sRcyText:='An Error Was Encountered While Trying To Close File. Please Contact Nutek For A Possible Solution.'),(sAlmText:='File Open Error While Deleting',sRcyText:='An Error Was Encountered While Trying To Open File. Please Contact Nutek For A Possible Solution.'),(sAlmText:='File Create Error While Deleting',sRcyText:='An Error Was Encountered While Trying To Create File. Please Contact Nutek For A Possible Solution.'),(sAlmText:='File Write Error While Deleting',sRcyText:='An Error Was Encountered While Trying To Write File. Please Contact Nutek For A Possible Solution.'),(sAlmText:='File Close Error While Deleting',sRcyText:='An Error Was Encountered While Trying To Close File. Please Contact Nutek For A Possible Solution.'),(sAlmText:='File Open Error While Getting List',sRcyText:='An Error Was Encountered While Trying To Open File. Please Contact Nutek For A Possible Solution.'),(sAlmText:='File Read Error While Getting List',sRcyText:='An Error Was Encountered While Trying To Read File. Please Contact Nutek For A Possible Solution.'),(sAlmText:='File Close Error While Getting List',sRcyText:='An Error Was Encountered While Trying To Close File. Please Contact Nutek For A Possible Solution.'),(sAlmText:='Directory Does Not Exist While Adding & Editing',sRcyText:='The Directory Does Not Exist.Please Contact Nutek For A Possible Solution.'),(sAlmText:='Directory Does Not Exist While Deleting',sRcyText:='The Directory Does Not Exist.Please Contact Nutek For A Possible Solution.'),(sAlmText:='File Open Error While Adding',sRcyText:='An Error Was Encountered While Trying To Open File. Please Contact Nutek For A Possible Solution.'),(sAlmText:='File Create Error While Adding',sRcyText:='An Error Was Encountered While Trying To Create File. Please Contact Nutek For A Possible Solution.'),(sAlmText:='File Write Error While Adding',sRcyText:='An Error Was Encountered While Trying To Write File. Please Contact Nutek For A Possible Solution.'),(sAlmText:='File Close Error While Adding',sRcyText:='An Error Was Encountered While Trying To Close File. Please Contact Nutek For A Possible Solution.'),(sAlmText:='Directory Does Not Exist While Adding',sRcyText:='The Directory Does Not Exist.Please Contact Nutek For A Possible Solution.'),(sAlmText:='File Open Error While Editing',sRcyText:='An Error Was Encountered While Trying To Open File. Please Contact Nutek For A Possible Solution.'),(sAlmText:='File Create Error While Editing',sRcyText:='An Error Was Encountered While Trying To Create File. Please Contact Nutek For A Possible Solution.'),(sAlmText:='File Write Error While Editing',sRcyText:='An Error Was Encountered While Trying To Write File. Please Contact Nutek For A Possible Solution.'),(sAlmText:='File Close Error While Editing',sRcyText:='An Error Was Encountered While Trying To Close File. Please Contact Nutek For A Possible Solution.'),(sAlmText:='Directory Does Not Exist While Editing',sRcyText:='The Directory Does Not Exist.Please Contact Nutek For A Possible Solution.'),(sAlmText:='File Open Error While Loading Current Recipe',sRcyText:='An Error Was Encountered While Trying To Open File. Please Contact Nutek For A Possible Solution.'),(sAlmText:='File Create Error While Loading Current Recipe',sRcyText:='An Error Was Encountered While Trying To Create File. Please Contact Nutek For A Possible Solution.'),(sAlmText:='File Write Error While Loading Current Recipe',sRcyText:='An Error Was Encountered While Trying To Write File. Please Contact Nutek For A Possible Solution.'),(sAlmText:='File Close Error While Loading Current Recipe',sRcyText:='An Error Was Encountered While Trying To Close File. Please Contact Nutek For A Possible Solution.'),(sAlmText:='Directory Does Not Exist While Loading Current Recipe',sRcyText:='The Directory Does Not Exist.Please Contact Nutek For A Possible Solution.'),(sAlmText:='File Open Error While Reading Current Recipe',sRcyText:='An Error Was Encountered While Trying To Open File. Please Contact Nutek For A Possible Solution.'),(sAlmText:='File Read Error While Reading Current Recipe',sRcyText:='An Error Was Encountered While Trying To Read File. Please Contact Nutek For A Possible Solution.'),(sAlmText:='File Close Error While Reading Current Recipe',sRcyText:='An Error Was Encountered While Trying To Close File. Please Contact Nutek For A Possible Solution.'),(sAlmText:='File Open Error While Writing Current Recipe Parameter',sRcyText:='An Error Was Encountered While Trying To Open File. Please Contact Nutek For A Possible Solution.'),(sAlmText:='File Create Error While Writing Current Recipe Parameter',sRcyText:='An Error Was Encountered While Trying To Create File. Please Contact Nutek For A Possible Solution.'),(sAlmText:='File Write Error While Writing Current Recipe Parameter',sRcyText:='An Error Was Encountered While Trying To Write File. Please Contact Nutek For A Possible Solution.'),(sAlmText:='File Close Error While Writing Current Recipe Parameter',sRcyText:='An Error Was Encountered While Trying To Close File. Please Contact Nutek For A Possible Solution.'),(sAlmText:='Directory Does Not Exist While Writing Current Recipe Parameter',sRcyText:='The Directory Does Not Exist.Please Contact Nutek For A Possible Solution.'),(sAlmText:='File Open Error While Writing Saving List',sRcyText:='An Error Was Encountered While Trying To Open File. Please Contact Nutek For A Possible Solution.'),(sAlmText:='File Create Error While Writing Saving List',sRcyText:='An Error Was Encountered While Trying To Create File. Please Contact Nutek For A Possible Solution.'),(sAlmText:='File Write Error While Writing Saving List',sRcyText:='An Error Was Encountered While Trying To Write File. Please Contact Nutek For A Possible Solution.'),(sAlmText:='File Close Error While Writing Saving List',sRcyText:='An Error Was Encountered While Trying To Close File. Please Contact Nutek For A Possible Solution.'),(sAlmText:='Directory Does Not Exist While Writing Saving List',sRcyText:='The Directory Does Not Exist.Please Contact Nutek For A Possible Solution.'),57(0)];
END_VAR
(**)
(*Local Output*)
VAR
	bNmExist : BOOL;
	bNmNotExist : BOOL;
	bNmEmpty : BOOL;
	bListFull : BOOL;
	sDebug : STRING[300];
	tyTempRecipe : tyProdRcpParam;
	a_tyCurrList : ARRAY[1..c_udiProdRcpMax] OF tyProdRcpParam;
	a_tyFilterList : ARRAY[1..c_udiProdRcpMax] OF tyProdRcpParam;
	a_tySortList : ARRAY[1..c_udiProdRcpMax] OF tyProdRcpParam;
	a_tyScanList : ARRAY[1..c_udiProdRcpMax] OF tyProdRcpParam;
	tyInfoOut : tyProdRcpParam;
	bFileNotFound : BOOL;
	a_tyCurrRcp : ARRAY[0..5] OF tyProdRcpParam;
	a_tyCurrZ2Rcp : ARRAY[0..5] OF tyProdRcpParam;
	iFilterCtr : INT;
END_VAR
(**)
(*Local Input*)
VAR
	udiRstErr : UDINT := 0;
	dtCurrDT : DATE_AND_TIME;
	sSearch : STRING[254] := '';
	sScan : STRING[254] := '';
	tyInfoIn : tyProdRcpParam;
	tyCurrRcpWr : tyProdRcpParam;
	sListFileName : STRING[80] := 'ProductRecipeList.dat';
	sSingleFileName : STRING[80] := 'ProductRecipe.dat';
	sProgNm : STRING[15] := 'ProdRcp';
	bNtSettingsLoadDone : BOOL := TRUE;
	bWidth2Prep : BOOL;
	uiSortNo : UDINT := 0;
END_VAR
(**)
(*Local*)
VAR
	sEndRcpName : STRING[254];
	bCreateRcp : BOOL;
	udiSortCurrenTotalCntr : UDINT;
	iSortCurrentInnerCntr : INT;
	iSortCurrentOuterCntr : INT;
	iTotalRcp : INT;
	udi : UDINT;
	bRstErr : BOOL;
	udiRstErrOld : UDINT;
	bInitDone : BOOL;
	bInitialDone : BOOL;
	usiStep : USINT;
	udiAddStatus : UDINT;
	a_tyListTemp : ARRAY[1..c_udiProdRcpMax] OF tyProdRcpParam;
	fbDirCreate1 : fbDirCreate;
	fbDirCreate2 : fbDirCreate;
	fbFileReadList : fbFileFullRead;
	fbFileWriteList : fbFileFullWrite;
	fbFileReadSingle : fbFileFullRead;
	fbFileLoadSingle : fbFileFullWrite;
	fbFileWriteSingle : fbFileFullWrite;
	udiModuleNum : UDINT := 4801;
END_VAR
```

#### InputRef_Link.var - not listed in the package file held
```iecst
(*2019-04-24*)
(**)
VAR
	rWidthInMM : REAL;
	rWidthInMM2 : REAL;
	sWidthInMM : STRING[30];
	sWidthInMM2 : STRING[30];
	p_bLinkStartupRun : REFERENCE TO BOOL;
	p_bLinkNtParamLCSManageRcpPrep : REFERENCE TO BOOL;
	p_bLinkMcParamLCSManageRcpEn : REFERENCE TO BOOL;
	p_eLinkLCSMngRcpProdRcpAct : REFERENCE TO eProdRcpAction;
	p_eLinkUIProdRcpAct : REFERENCE TO eProdRcpAction;
END_VAR
```

#### Act_InitGlobal.st - not listed in the package file held
```iecst
(** 2020-06-08 **)
ACTION Act_InitGlobal:

	(* Always Change If Project Change *)

	//Pass Data To Link
	p_bLinkStartupRun ACCESS p_StartupRun;
	p_bLinkNtParamLCSManageRcpPrep ACCESS p_NtParamLCSManageRcpPrep;
	p_bLinkMcParamLCSManageRcpEn ACCESS p_McParamLCSManageRcpEn;
	p_eLinkLCSMngRcpProdRcpAct ACCESS p_LCSMngRcpProdRcpAct;
	p_eLinkUIProdRcpAct ACCESS p_UIProdRcpAct;

	//Pass Data To Internal Use
	p_udiRstErr ACCESS p_RstErrReset;
	p_dtCurrDT ACCESS p_TimeCurrDT;
	p_sSearch ACCESS p_UIProdRcpSearch;
	p_tyInfoIn ACCESS p_UIProdRcpInfoIn;
	p_tyCurrRcpWr ACCESS p_UIProdRcpCurrRcpWr;
	p_sListFileName ACCESS p_NtParamProdRcpListFileNm;
	p_sSingleFileName ACCESS p_NtParamProdRcpSingleFileNm;
	p_sProgNm ACCESS p_NtParamProdRcpProgNm;
	p_bNtSettingsLoadDone ACCESS p_StartupNtSettingsLoadDone;
	p_bWidth2Prep ACCESS p_NtParamLFWidth2Prep;
	(* Always Change If Project Change *)

END_ACTION
```

#### Act_Link.st - not listed in the package file held
```iecst
(** 2019-04-30 **)
ACTION Act_Link:

	IF (p_eAct = ProdRcpActAddEdit) OR (p_eAct = ProdRcpActAdd) OR (p_eAct = ProdRcpActEdit) THEN

		rWidthInMM				:= DINT_TO_REAL(p_tyInfoIn.diWidthInUM);
		rWidthInMM2				:= DINT_TO_REAL(p_tyInfoIn.diWidthInUM2);
		rWidthInMM				:= rWidthInMM / 1000;
		rWidthInMM2				:= rWidthInMM2 / 1000;
		sWidthInMM				:= REAL_TO_STRING(rWidthInMM);
		sWidthInMM2				:= REAL_TO_STRING(rWidthInMM2);

		IF p_bWidth2Prep THEN
			p_tyInfoIn.sDisplayInfo	:= sWidthInMM;
			p_tyInfoIn.sDisplayInfo	:= CONCAT(p_tyInfoIn.sDisplayInfo , ' | ');
			p_tyInfoIn.sDisplayInfo	:= CONCAT(p_tyInfoIn.sDisplayInfo , sWidthInMM2);
			p_tyInfoIn.sDisplayInfo	:= CONCAT(p_tyInfoIn.sDisplayInfo , ' mm');
		ELSE
			p_tyInfoIn.sDisplayInfo	:= sWidthInMM;
			p_tyInfoIn.sDisplayInfo	:= CONCAT(p_tyInfoIn.sDisplayInfo , ' mm');
		END_IF

	END_IF

END_ACTION
```

### MpProdRcp.typ - Change By Project
```iecst
(*2019-04-28*)
(**)
(*Action*)

TYPE
	eMpProdRcpAction :
		(
		MpProdRcpActIdle,
		MpProdRcpActCreateDir,
		MpProdRcpActLoad,
		MpProdRcpActSave
		);
	tyMpProdRcp : 	STRUCT
		In : tyMpProdRcpIn1;
		Out : tyMpProdRcpOut1;
	END_STRUCT;
	tyMpProdRcpIn1 : 	STRUCT
		eAct : eMpProdRcpAction;
		tyMpProdRcpMpLink : MpComIdentType;
		sPVName : STRING[100];
		sFileName : STRING[255];
		sProgNm : STRING[15];
		bNtSettingsLoadDone : BOOL;
		udiRstErr : UDINT;
	END_STRUCT;
	tyMpProdRcpOut1 : 	STRUCT
		eStat : eMpProdRcpAction;
		eStatus : eFBStatus;
		sStatTxt : STRING[200];
		tyAlmData : tyAlmDat;
	END_STRUCT;
END_TYPE
```

### MpProdRcp.var - Change By Project
```iecst
VAR
	g_tyMpProdRcp : tyMpProdRcpOut1;
END_VAR
```

### Program Logical/MpProdRcp/MpProdRcp (IEC) - 1.00.0 - NtRecipe v5.00.0 , NtFileIO v5.00.0

#### Local.var
```iecst
VAR
	tylocalMpProdRcp : tyMpProdRcp;
	pa_tyMpProdRcp : REFERENCE TO ARRAY[0..c_udiMpProdRcpMax] OF tyProdRcpParam;
	udiStatus : UDINT := 0;
	sStatTxt : STRING[200] := '';
	a_sStatText : ARRAY[0..50] OF STRING[200] := ['Idling','Creating Directory','Loading Mp Product Recipe','Saving Mp Product Recipe',47('')];
END_VAR
(**)
(*Local Alarm*)
VAR
	tyAlmData : tyAlmDat;
END_VAR
(**)
VAR
	udiRstErr : UDINT := 0;
	a_tyMpProdRcp : ARRAY[0..c_udiMpProdRcpMax] OF tyProdRcpParam;
	tyMpProdRcpMpLink : MpComIdentType;
	sPVName : STRING[100] := 'MpProdRcp:a_tyMpProdRcp1';
	sFileName : STRING[255] := 'MpProductRecipe.xml';
	sProgNm : STRING[15] := 'MpProdRcp';
	bNtSettingsLoadDone : BOOL := TRUE;
END_VAR
(**)
(*Local*)
VAR
	bRstErr : BOOL;
	udiRstErrOld : UDINT;
	bInitDone : BOOL;
	bInitialDone : BOOL;
	usiStep : USINT;
	a_tyMpProdRcp1 : ARRAY[0..c_udiMpProdRcpMax] OF tyProdRcpParam;
	fbDirCreate1 : fbDirCreate;
	fbDirCreate2 : fbDirCreate;
	fbMpRecipeRegPar : MpRecipeRegPar;
	fbMpRecipeXml : MpRecipeXml;
END_VAR
VAR CONSTANT
	c_udiMpProdRcpMax : UDINT := 1999;
END_VAR
VAR
	udiModuleNum : UDINT := 5001;
END_VAR
```

#### Act_Alarm.st
```iecst
ACTION Act_Alarm:

	IF tylocalMpProdRcp.In.udiRstErr <> udiRstErrOld THEN
		bRstErr			:= TRUE;
		udiRstErrOld	:= tylocalMpProdRcp.In.udiRstErr;
	ELSE
		bRstErr			:= FALSE;
	END_IF

	//Reset Error
	IF (tylocalMpProdRcp.Out.eStatus = Error) AND bRstErr THEN
		tylocalMpProdRcp.In.eAct	:= MpProdRcpActIdle;
		tylocalMpProdRcp.Out.eStat	:= MpProdRcpActIdle;
	END_IF

	//Reset Done
	IF tylocalMpProdRcp.Out.eStatus = Done AND tylocalMpProdRcp.In.eAct = MpProdRcpActIdle THEN
		tylocalMpProdRcp.Out.eStat	:= MpProdRcpActIdle;
	END_IF

	//Error
	IF EDGEPOS(tylocalMpProdRcp.Out.eStatus = Error) THEN

		tylocalMpProdRcp.Out.tyAlmData.udiCode		:= udiStatus;
		tylocalMpProdRcp.Out.tyAlmData.eSeverity	:= AlmSeverityError;
		tylocalMpProdRcp.Out.tyAlmData.udiRunTime	:= tylocalMpProdRcp.Out.tyAlmData.udiRunTime + 1;
		tylocalMpProdRcp.Out.tyAlmData.bAlm			:= TRUE;
		tylocalMpProdRcp.Out.tyAlmData.udiModuleNum	:= udiModuleNum;
		g_tyAlmProgNm.sMpProdRcpProgNm				:= tylocalMpProdRcp.In.sProgNm;

	ELSIF bRstErr AND (tylocalMpProdRcp.Out.tyAlmData.udiCode <> 0) THEN

		tylocalMpProdRcp.Out.tyAlmData.udiCode		:= 0;
		tylocalMpProdRcp.Out.tyAlmData.eSeverity	:= AlmSeverityNA;
		tylocalMpProdRcp.Out.tyAlmData.bAlm			:= FALSE;

		sStatTxt	:= a_sStatText[tylocalMpProdRcp.Out.eStat];

	END_IF

END_ACTION
```

#### Act_Initial.st
```iecst
(** 2019-04-28 **)
ACTION Act_Initial:

	//Initial
	sStatTxt	:= a_sStatText[tylocalMpProdRcp.Out.eStat];

	fbDirCreate1.sDevice	:= 'F';
	fbDirCreate1.sDirName	:= 'User';
	fbDirCreate1(bEn := FALSE);

	fbDirCreate2.sDevice	:= 'User';
	fbDirCreate2.sDirName	:= 'ProductRecipeXml';
	fbDirCreate2(bEn := FALSE);

	tylocalMpProdRcp.In.tyMpProdRcpMpLink	:= gRecipeXml;

	fbMpRecipeRegPar.MpLink	:= ADR(tylocalMpProdRcp.In.tyMpProdRcpMpLink);
	fbMpRecipeRegPar.PVName	:= ADR(tylocalMpProdRcp.In.sPVName);
	fbMpRecipeRegPar(Enable := FALSE);

	fbMpRecipeXml.MpLink		:= ADR(tylocalMpProdRcp.In.tyMpProdRcpMpLink);
	fbMpRecipeXml.DeviceName	:= ADR('MpProdRcp');
	fbMpRecipeXml.FileName		:= ADR(tylocalMpProdRcp.In.sFileName);
	fbMpRecipeXml(Enable := FALSE);

END_ACTION
```
